LIN {X 0,Y 362,Z 148.389,A -85,B 0,C 180,E1 -12973.899,E2 -12973.899} C_VEL
LIN {X 0,Y 361.929,Z 148.396,A -85,B 0,C 180,E1 -12976.934,E2 -12976.934} C_VEL
LIN {X 0,Y 361.889,Z 148.404,A -85,B 0,C 180,E1 -12980.461,E2 -12980.461} C_VEL
LIN {X 0,Y 361.895,Z 148.403,A -85,B 0,C 180,E1 -12984.113,E2 -12984.113} C_VEL
LIN {X 0,Y 361.844,Z 148.41,A -85,B 0,C 180,E1 -12987.785,E2 -12987.785} C_VEL
LIN {X 0,Y 361.849,Z 148.409,A -85,B 0,C 180,E1 -12991.285,E2 -12991.285} C_VEL
LIN {X 0,Y 361.856,Z 148.405,A -85,B 0,C 180,E1 -12994.28,E2 -12994.28} C_VEL
LIN {X 0,Y 361.862,Z 148.405,A -85,B 0,C 180,E1 -12997.222,E2 -12997.222} C_VEL
LIN {X 0,Y 361.815,Z 148.415,A -85,B 0,C 180,E1 -13000.751,E2 -13000.751} C_VEL
LIN {X 0,Y 361.819,Z 148.419,A -85,B 0,C 180,E1 -13004.369,E2 -13004.369} C_VEL
LIN {X 0,Y 361.838,Z 148.415,A -85,B 0,C 180,E1 -13007.568,E2 -13007.568} C_VEL
LIN {X 0,Y 361.868,Z 148.41,A -85,B 0,C 180,E1 -13010.974,E2 -13010.974} C_VEL
LIN {X 0,Y 361.877,Z 148.405,A -85,B 0,C 180,E1 -13014.655,E2 -13014.655} C_VEL
LIN {X 0,Y 361.897,Z 148.548,A -85,B 0,C 180,E1 -13018.09,E2 -13018.09} C_VEL
LIN {X 0,Y 364.754,Z 160.107,A -85,B 0,C 180,E1 -13021.204,E2 -13021.204} C_VEL
LIN {X 0,Y 366.747,Z 170.569,A -85,B 0,C 180,E1 -13023.848,E2 -13023.848} C_VEL
LIN {X 0,Y 366.502,Z 174.041,A -85,B 0,C 180,E1 -13024.632,E2 -13024.632} C_VEL
LIN {X 0,Y 365.411,Z 184.836,A -85,B 0,C 180,E1 -13026.971,E2 -13026.971} C_VEL
LIN {X 0,Y 369.803,Z 207.145,A -85,B 0,C 180,E1 -13027.794,E2 -13027.794} C_VEL
LIN {X 0,Y 371.958,Z 222.29,A -85,B 0,C 180,E1 -13028.279,E2 -13028.279} C_VEL
LIN {X 0,Y 370.513,Z 294.23,A -85,B 0,C 180,E1 -13029.746,E2 -13029.746} C_VEL
LIN {X 0,Y 369.669,Z 307.871,A -85,B 0,C 180,E1 -13030.242,E2 -13030.242} C_VEL
LIN {X 0,Y 368.714,Z 319.646,A -85,B 0,C 180,E1 -13030.876,E2 -13030.876} C_VEL
LIN {X 0,Y 367.504,Z 331.641,A -85,B 0,C 180,E1 -13031.751,E2 -13031.751} C_VEL
LIN {X 0,Y 366.177,Z 343.107,A -85,B 0,C 180,E1 -13032.837,E2 -13032.837} C_VEL
LIN {X 0,Y 364.898,Z 353.468,A -85,B 0,C 180,E1 -13034.07,E2 -13034.07} C_VEL
LIN {X 0,Y 363.679,Z 362.827,A -85,B 0,C 180,E1 -13035.45,E2 -13035.45} C_VEL
LIN {X 0,Y 362.617,Z 371.909,A -85,B 0,C 180,E1 -13037.121,E2 -13037.121} C_VEL
LIN {X 0,Y 361.598,Z 379.26,A -85,B 0,C 180,E1 -13038.792,E2 -13038.792} C_VEL
LIN {X 0,Y 361.014,Z 385.178,A -85,B 0,C 180,E1 -13040.475,E2 -13040.475} C_VEL
LIN {X 0,Y 360.643,Z 389.866,A -85,B 0,C 180,E1 -13042.16,E2 -13042.16} C_VEL
LIN {X 0,Y 360.424,Z 393.696,A -85,B 0,C 180,E1 -13043.97,E2 -13043.97} C_VEL
LIN {X 0,Y 360.363,Z 396.045,A -85,B 0,C 180,E1 -13045.526,E2 -13045.526} C_VEL
LIN {X 0,Y 360.325,Z 397.269,A -85,B 0,C 180,E1 -13046.645,E2 -13046.645} C_VEL
LIN {X 0,Y 360.456,Z 398.443,A -85,B 0,C 180,E1 -13048.883,E2 -13048.883} C_VEL
LIN {X 0,Y 360.482,Z 398.443,A -85,B 0,C 180,E1 -13050,E2 -13050} C_VEL
LIN {X 0,Y 360.477,Z 398.05,A -85,B 0,C 180,E1 -13051.117,E2 -13051.117} C_VEL
LIN {X 0,Y 360.392,Z 397.212,A -85,B 0,C 180,E1 -13052.235,E2 -13052.235} C_VEL
LIN {X 0,Y 360.394,Z 394.304,A -85,B 0,C 180,E1 -13054.474,E2 -13054.474} C_VEL
LIN {X 0,Y 360.378,Z 391.384,A -85,B 0,C 180,E1 -13055.961,E2 -13055.961} C_VEL
LIN {X 0,Y 360.595,Z 386.495,A -85,B 0,C 180,E1 -13057.841,E2 -13057.841} C_VEL
LIN {X 0,Y 360.911,Z 380.822,A -85,B 0,C 180,E1 -13059.527,E2 -13059.527} C_VEL
LIN {X 0,Y 361.428,Z 373.709,A -85,B 0,C 180,E1 -13061.212,E2 -13061.212} C_VEL
LIN {X 0,Y 362.252,Z 364.807,A -85,B 0,C 180,E1 -13062.892,E2 -13062.892} C_VEL
LIN {X 0,Y 363.035,Z 356.181,A -85,B 0,C 180,E1 -13064.216,E2 -13064.216} C_VEL
LIN {X 0,Y 363.926,Z 345.713,A -85,B 0,C 180,E1 -13065.528,E2 -13065.528} C_VEL
LIN {X 0,Y 364.892,Z 334.368,A -85,B 0,C 180,E1 -13066.648,E2 -13066.648} C_VEL
LIN {X 0,Y 365.857,Z 321.79,A -85,B 0,C 180,E1 -13067.611,E2 -13067.611} C_VEL
LIN {X 0,Y 366.732,Z 308.962,A -85,B 0,C 180,E1 -13068.325,E2 -13068.325} C_VEL
LIN {X 0,Y 367.348,Z 295.296,A -85,B 0,C 180,E1 -13068.835,E2 -13068.835} C_VEL
LIN {X 0,Y 368.207,Z 245.144,A -85,B 0,C 180,E1 -13069.854,E2 -13069.854} C_VEL
LIN {X 0,Y 368.459,Z 220.259,A -85,B 0,C 180,E1 -13070.35,E2 -13070.35} C_VEL
LIN {X 0,Y 363.754,Z 185.456,A -85,B 0,C 180,E1 -13071.313,E2 -13071.313} C_VEL
LIN {X 0,Y 365.115,Z 169.471,A -85,B 0,C 180,E1 -13074.75,E2 -13074.75} C_VEL
LIN {X 0,Y 365.237,Z 165.158,A -85,B 0,C 180,E1 -13075.698,E2 -13075.698} C_VEL
LIN {X 0,Y 362.523,Z 151.236,A -85,B 0,C 180,E1 -13078.99,E2 -13078.99} C_VEL
LIN {X 0,Y 361.908,Z 148.408,A -85,B 0,C 180,E1 -13079.696,E2 -13079.696} C_VEL
LIN {X 0,Y 361.862,Z 148.407,A -85,B 0,C 180,E1 -13083.369,E2 -13083.369} C_VEL
LIN {X 0,Y 361.869,Z 148.406,A -85,B 0,C 180,E1 -13087.018,E2 -13087.018} C_VEL
LIN {X 0,Y 361.856,Z 148.413,A -85,B 0,C 180,E1 -13089.861,E2 -13089.861} C_VEL
LIN {X 0,Y 361.837,Z 148.41,A -85,B 0,C 180,E1 -13092.828,E2 -13092.828} C_VEL
LIN {X 0,Y 361.819,Z 148.415,A -85,B 0,C 180,E1 -13095.946,E2 -13095.946} C_VEL
LIN {X 0,Y 361.836,Z 148.412,A -85,B 0,C 180,E1 -13099.244,E2 -13099.244} C_VEL
LIN {X 0,Y 361.863,Z 148.407,A -85,B 0,C 180,E1 -13102.777,E2 -13102.777} C_VEL
LIN {X 0,Y 361.854,Z 148.411,A -85,B 0,C 180,E1 -13105.719,E2 -13105.719} C_VEL
LIN {X 0,Y 361.875,Z 148.408,A -85,B 0,C 180,E1 -13109.672,E2 -13109.672} C_VEL
LIN {X 0,Y 361.955,Z 148.399,A -85,B 0,C 180,E1 -13113.475,E2 -13113.475} C_VEL
LIN {X 0,Y 361.883,Z 148.41,A -85,B 0,C 180,E1 -13117.144,E2 -13117.144} C_VEL
LIN {X 0,Y 361.886,Z 148.406,A -85,B 0,C 180,E1 -13120.722,E2 -13120.722} C_VEL
LIN {X 0,Y 361.943,Z 148.396,A -85,B 0,C 180,E1 -13124.226,E2 -13124.226} C_VEL
LIN {X 0,Y 361.999,Z 148.391,A -85,B 0,C 180,E1 -13126.528,E2 -13126.528} C_VEL
LIN {X 0,Y 362,Z 148.389,A -85,B 0,C 180,E1 -13129.937,E2 -13129.937} C_VEL
LIN {X 0,Y 362.135,Z 148.374,A -85,B 0,C 180,E1 -13133.313,E2 -13133.313} C_VEL
LIN {X 0,Y 362.281,Z 148.354,A -85,B 0,C 180,E1 -13137.776,E2 -13137.776} C_VEL
LIN {X 0,Y 362.426,Z 148.337,A -85,B 0,C 180,E1 -13140,E2 -13140} C_VEL
LIN {X 0,Y 362.282,Z 148.356,A -85,B 0,C 180,E1 -13142.223,E2 -13142.223} C_VEL
LIN {X 0,Y 362.16,Z 148.374,A -85,B 0,C 180,E1 -13146.686,E2 -13146.686} C_VEL
LIN {X 0,Y 362.031,Z 148.388,A -85,B 0,C 180,E1 -13150.062,E2 -13150.062} C_VEL
LIN {X 0,Y 361.997,Z 148.391,A -85,B 0,C 180,E1 -13153.899,E2 -13153.899} C_VEL
LIN {X 0,Y 361.966,Z 148.396,A -85,B 0,C 180,E1 -13157.938,E2 -13157.938} C_VEL
LIN {X 0,Y 361.861,Z 148.408,A -85,B 0,C 180,E1 -13161.655,E2 -13161.655} C_VEL
LIN {X 0,Y 361.926,Z 148.399,A -85,B 0,C 180,E1 -13165.29,E2 -13165.29} C_VEL
LIN {X 0,Y 361.907,Z 148.404,A -85,B 0,C 180,E1 -13167.779,E2 -13167.779} C_VEL
LIN {X 0,Y 361.837,Z 148.412,A -85,B 0,C 180,E1 -13171.629,E2 -13171.629} C_VEL
LIN {X 0,Y 361.873,Z 148.406,A -85,B 0,C 180,E1 -13175.345,E2 -13175.345} C_VEL
LIN {X 0,Y 361.869,Z 148.406,A -85,B 0,C 180,E1 -13179.027,E2 -13179.027} C_VEL
LIN {X 0,Y 361.835,Z 148.41,A -85,B 0,C 180,E1 -13182.829,E2 -13182.829} C_VEL
LIN {X 0,Y 361.817,Z 148.415,A -85,B 0,C 180,E1 -13185.947,E2 -13185.947} C_VEL
LIN {X 0,Y 361.834,Z 148.413,A -85,B 0,C 180,E1 -13189.245,E2 -13189.245} C_VEL
LIN {X 0,Y 361.862,Z 148.407,A -85,B 0,C 180,E1 -13192.777,E2 -13192.777} C_VEL
LIN {X 0,Y 361.853,Z 148.411,A -85,B 0,C 180,E1 -13195.72,E2 -13195.72} C_VEL
LIN {X 0,Y 361.874,Z 148.408,A -85,B 0,C 180,E1 -13199.672,E2 -13199.672} C_VEL
LIN {X 0,Y 361.954,Z 148.399,A -85,B 0,C 180,E1 -13203.475,E2 -13203.475} C_VEL
LIN {X 0,Y 361.882,Z 148.41,A -85,B 0,C 180,E1 -13207.144,E2 -13207.144} C_VEL
LIN {X 0,Y 361.885,Z 148.406,A -85,B 0,C 180,E1 -13210.722,E2 -13210.722} C_VEL
LIN {X 0,Y 361.943,Z 148.397,A -85,B 0,C 180,E1 -13214.226,E2 -13214.226} C_VEL
LIN {X 0,Y 361.999,Z 148.392,A -85,B 0,C 180,E1 -13216.528,E2 -13216.528} C_VEL
LIN {X 0,Y 362,Z 148.389,A -85,B 0,C 180,E1 -13219.937,E2 -13219.937} C_VEL
LIN {X 0,Y 362.135,Z 148.374,A -85,B 0,C 180,E1 -13223.313,E2 -13223.313} C_VEL
LIN {X 0,Y 362.171,Z 148.447,A -85,B 0,C 180,E1 -13227.08,E2 -13227.08} C_VEL
LIN {X 0,Y 363.379,Z 154.733,A -85,B 0,C 180,E1 -13228.771,E2 -13228.771} C_VEL
LIN {X 0,Y 366.752,Z 166.026,A -85,B 0,C 180,E1 -13229.179,E2 -13229.179} C_VEL
LIN {X 0,Y 369.104,Z 178.936,A -85,B 0,C 180,E1 -13229.56,E2 -13229.56} C_VEL
LIN {X 0,Y 367.632,Z 262.636,A -85,B 0,C 180,E1 -13231.233,E2 -13231.233} C_VEL
LIN {X 0,Y 367.191,Z 276.354,A -85,B 0,C 180,E1 -13231.748,E2 -13231.748} C_VEL
LIN {X 0,Y 366.675,Z 288.171,A -85,B 0,C 180,E1 -13232.403,E2 -13232.403} C_VEL
LIN {X 0,Y 365.891,Z 300.242,A -85,B 0,C 180,E1 -13233.304,E2 -13233.304} C_VEL
LIN {X 0,Y 365.039,Z 311.767,A -85,B 0,C 180,E1 -13234.417,E2 -13234.417} C_VEL
LIN {X 0,Y 364.12,Z 322.178,A -85,B 0,C 180,E1 -13235.677,E2 -13235.677} C_VEL
LIN {X 0,Y 363.128,Z 332.343,A -85,B 0,C 180,E1 -13237.227,E2 -13237.227} C_VEL
LIN {X 0,Y 362.301,Z 341.262,A -85,B 0,C 180,E1 -13238.928,E2 -13238.928} C_VEL
LIN {X 0,Y 361.648,Z 348.361,A -85,B 0,C 180,E1 -13240.639,E2 -13240.639} C_VEL
LIN {X 0,Y 361.152,Z 354.036,A -85,B 0,C 180,E1 -13242.361,E2 -13242.361} C_VEL
LIN {X 0,Y 360.805,Z 358.477,A -85,B 0,C 180,E1 -13244.092,E2 -13244.092} C_VEL
LIN {X 0,Y 360.509,Z 361.81,A -85,B 0,C 180,E1 -13245.839,E2 -13245.839} C_VEL
LIN {X 0,Y 360.358,Z 363.616,A -85,B 0,C 180,E1 -13247.131,E2 -13247.131} C_VEL
LIN {X 0,Y 360.286,Z 364.645,A -85,B 0,C 180,E1 -13248.186,E2 -13248.186} C_VEL
LIN {X 0,Y 360.274,Z 365.465,A -85,B 0,C 180,E1 -13249.708,E2 -13249.708} C_VEL
LIN {X 0,Y 360.311,Z 365.692,A -85,B 0,C 180,E1 -13250.568,E2 -13250.568} C_VEL
LIN {X 0,Y 360.34,Z 365.549,A -85,B 0,C 180,E1 -13251.751,E2 -13251.751} C_VEL
LIN {X 0,Y 360.522,Z 364.413,A -85,B 0,C 180,E1 -13253.621,E2 -13253.621} C_VEL
LIN {X 0,Y 360.663,Z 363.388,A -85,B 0,C 180,E1 -13254.55,E2 -13254.55} C_VEL
LIN {X 0,Y 360.166,Z 362.258,A -85,B 0,C 180,E1 -13255.467,E2 -13255.467} C_VEL
LIN {X 0,Y 357.686,Z 359.944,A -85,B 0,C 180,E1 -13256.956,E2 -13256.956} C_VEL
LIN {X 0,Y 355.646,Z 357.657,A -85,B 0,C 180,E1 -13258.138,E2 -13258.138} C_VEL
LIN {X 0,Y 354.922,Z 355.563,A -85,B 0,C 180,E1 -13259.026,E2 -13259.026} C_VEL
LIN {X 0,Y 354.946,Z 354.762,A -85,B 0,C 180,E1 -13259.319,E2 -13259.319} C_VEL
LIN {X 0,Y 355.694,Z 349.778,A -85,B 0,C 180,E1 -13260.912,E2 -13260.912} C_VEL
LIN {X 0,Y 356.802,Z 342.363,A -85,B 0,C 180,E1 -13262.798,E2 -13262.798} C_VEL
LIN {X 0,Y 358.029,Z 334.009,A -85,B 0,C 180,E1 -13264.468,E2 -13264.468} C_VEL
LIN {X 0,Y 359.219,Z 324.905,A -85,B 0,C 180,E1 -13265.94,E2 -13265.94} C_VEL
LIN {X 0,Y 360.637,Z 314.081,A -85,B 0,C 180,E1 -13267.341,E2 -13267.341} C_VEL
LIN {X 0,Y 362.038,Z 302.196,A -85,B 0,C 180,E1 -13268.534,E2 -13268.534} C_VEL
LIN {X 0,Y 363.121,Z 289.635,A -85,B 0,C 180,E1 -13269.515,E2 -13269.515} C_VEL
LIN {X 0,Y 363.912,Z 277.193,A -85,B 0,C 180,E1 -13270.223,E2 -13270.223} C_VEL
LIN {X 0,Y 364.539,Z 263.315,A -85,B 0,C 180,E1 -13270.752,E2 -13270.752} C_VEL
LIN {X 0,Y 366.444,Z 181.628,A -85,B 0,C 180,E1 -13272.428,E2 -13272.428} C_VEL
LIN {X 0,Y 365.137,Z 176.337,A -85,B 0,C 180,E1 -13272.647,E2 -13272.647} C_VEL
LIN {X 0,Y 357.636,Z 158.854,A -85,B 0,C 180,E1 -13273.66,E2 -13273.66} C_VEL
LIN {X 0,Y 356.429,Z 155.986,A -85,B 0,C 180,E1 -13273.846,E2 -13273.846} C_VEL
LIN {X 0,Y 354.78,Z 149.298,A -85,B 0,C 180,E1 -13275.91,E2 -13275.91} C_VEL
LIN {X 0,Y 354.765,Z 149.297,A -85,B 0,C 180,E1 -13279.176,E2 -13279.176} C_VEL
LIN {X 0,Y 354.799,Z 149.289,A -85,B 0,C 180,E1 -13282.405,E2 -13282.405} C_VEL
LIN {X 0,Y 354.808,Z 149.288,A -85,B 0,C 180,E1 -13284.941,E2 -13284.941} C_VEL
LIN {X 0,Y 354.793,Z 149.292,A -85,B 0,C 180,E1 -13288.406,E2 -13288.406} C_VEL
LIN {X 0,Y 354.797,Z 149.289,A -85,B 0,C 180,E1 -13291.615,E2 -13291.615} C_VEL
LIN {X 0,Y 354.804,Z 149.29,A -85,B 0,C 180,E1 -13295.42,E2 -13295.42} C_VEL
LIN {X 0,Y 354.816,Z 149.288,A -85,B 0,C 180,E1 -13299.113,E2 -13299.113} C_VEL
LIN {X 0,Y 354.837,Z 149.287,A -85,B 0,C 180,E1 -13302.717,E2 -13302.717} C_VEL
LIN {X 0,Y 354.909,Z 149.274,A -85,B 0,C 180,E1 -13306.254,E2 -13306.254} C_VEL
LIN {X 0,Y 354.949,Z 149.262,A -85,B 0,C 180,E1 -13309.735,E2 -13309.735} C_VEL
LIN {X 0,Y 355.088,Z 149.245,A -85,B 0,C 180,E1 -13313.18,E2 -13313.18} C_VEL
LIN {X 0,Y 355.22,Z 149.228,A -85,B 0,C 180,E1 -13317.732,E2 -13317.732} C_VEL
LIN {X 0,Y 355.146,Z 149.244,A -85,B 0,C 180,E1 -13321.134,E2 -13321.134} C_VEL
LIN {X 0,Y 355.227,Z 149.225,A -85,B 0,C 180,E1 -13322.268,E2 -13322.268} C_VEL
LIN {X 0,Y 355.089,Z 149.248,A -85,B 0,C 180,E1 -13326.82,E2 -13326.82} C_VEL
LIN {X 0,Y 354.956,Z 149.269,A -85,B 0,C 180,E1 -13330.265,E2 -13330.265} C_VEL
LIN {X 0,Y 354.945,Z 149.269,A -85,B 0,C 180,E1 -13334.019,E2 -13334.019} C_VEL
LIN {X 0,Y 354.892,Z 149.269,A -85,B 0,C 180,E1 -13338.092,E2 -13338.092} C_VEL
LIN {X 0,Y 354.821,Z 149.279,A -85,B 0,C 180,E1 -13341.418,E2 -13341.418} C_VEL
LIN {X 0,Y 354.851,Z 149.282,A -85,B 0,C 180,E1 -13344.577,E2 -13344.577} C_VEL
LIN {X 0,Y 354.802,Z 149.288,A -85,B 0,C 180,E1 -13348.386,E2 -13348.386} C_VEL
LIN {X 0,Y 354.789,Z 149.29,A -85,B 0,C 180,E1 -13352.333,E2 -13352.333} C_VEL
LIN {X 0,Y 354.824,Z 149.286,A -85,B 0,C 180,E1 -13355.699,E2 -13355.699} C_VEL
LIN {X 0,Y 354.77,Z 149.293,A -85,B 0,C 180,E1 -13359.413,E2 -13359.413} C_VEL
LIN {X 0,Y 354.787,Z 149.291,A -85,B 0,C 180,E1 -13362.867,E2 -13362.867} C_VEL
LIN {X 0,Y 354.769,Z 149.294,A -85,B 0,C 180,E1 -13366.104,E2 -13366.104} C_VEL
LIN {X 0,Y 354.788,Z 149.293,A -85,B 0,C 180,E1 -13369.179,E2 -13369.179} C_VEL
LIN {X 0,Y 354.808,Z 149.281,A -85,B 0,C 180,E1 -13372.403,E2 -13372.403} C_VEL
LIN {X 0,Y 354.814,Z 149.283,A -85,B 0,C 180,E1 -13374.941,E2 -13374.941} C_VEL
LIN {X 0,Y 354.841,Z 149.47,A -85,B 0,C 180,E1 -13377.588,E2 -13377.588} C_VEL
LIN {X 0,Y 357.879,Z 161.515,A -85,B 0,C 180,E1 -13380.92,E2 -13380.92} C_VEL
LIN {X 0,Y 359.925,Z 172.344,A -85,B 0,C 180,E1 -13383.718,E2 -13383.718} C_VEL
LIN {X 0,Y 358.686,Z 184.194,A -85,B 0,C 180,E1 -13386.412,E2 -13386.412} C_VEL
LIN {X 0,Y 363.396,Z 208.056,A -85,B 0,C 180,E1 -13387.327,E2 -13387.327} C_VEL
LIN {X 0,Y 365.533,Z 223.693,A -85,B 0,C 180,E1 -13387.835,E2 -13387.835} C_VEL
LIN {X 0,Y 364.043,Z 294.036,A -85,B 0,C 180,E1 -13389.296,E2 -13389.296} C_VEL
LIN {X 0,Y 363.162,Z 307.631,A -85,B 0,C 180,E1 -13389.799,E2 -13389.799} C_VEL
LIN {X 0,Y 362.112,Z 319.389,A -85,B 0,C 180,E1 -13390.44,E2 -13390.44} C_VEL
LIN {X 0,Y 360.948,Z 330.571,A -85,B 0,C 180,E1 -13391.26,E2 -13391.26} C_VEL
LIN {X 0,Y 359.569,Z 342.172,A -85,B 0,C 180,E1 -13392.364,E2 -13392.364} C_VEL
LIN {X 0,Y 358.176,Z 352.638,A -85,B 0,C 180,E1 -13393.617,E2 -13393.617} C_VEL
LIN {X 0,Y 357.081,Z 360.972,A -85,B 0,C 180,E1 -13394.843,E2 -13394.843} C_VEL
LIN {X 0,Y 356.081,Z 369.153,A -85,B 0,C 180,E1 -13396.299,E2 -13396.299} C_VEL
LIN {X 0,Y 354.91,Z 376.956,A -85,B 0,C 180,E1 -13397.999,E2 -13397.999} C_VEL
LIN {X 0,Y 354.186,Z 383.231,A -85,B 0,C 180,E1 -13399.712,E2 -13399.712} C_VEL
LIN {X 0,Y 353.691,Z 388.249,A -85,B 0,C 180,E1 -13401.429,E2 -13401.429} C_VEL
LIN {X 0,Y 353.397,Z 392.158,A -85,B 0,C 180,E1 -13403.147,E2 -13403.147} C_VEL
LIN {X 0,Y 353.274,Z 395.798,A -85,B 0,C 180,E1 -13405.436,E2 -13405.436} C_VEL
LIN {X 0,Y 353.244,Z 396.993,A -85,B 0,C 180,E1 -13406.578,E2 -13406.578} C_VEL
LIN {X 0,Y 353.358,Z 398.126,A -85,B 0,C 180,E1 -13408.86,E2 -13408.86} C_VEL
LIN {X 0,Y 353.4,Z 398.109,A -85,B 0,C 180,E1 -13410,E2 -13410} C_VEL
LIN {X 0,Y 353.38,Z 397.69,A -85,B 0,C 180,E1 -13411.139,E2 -13411.139} C_VEL
LIN {X 0,Y 353.294,Z 396.823,A -85,B 0,C 180,E1 -13412.28,E2 -13412.28} C_VEL
LIN {X 0,Y 353.261,Z 395.554,A -85,B 0,C 180,E1 -13413.421,E2 -13413.421} C_VEL
LIN {X 0,Y 353.261,Z 392.846,A -85,B 0,C 180,E1 -13415.136,E2 -13415.136} C_VEL
LIN {X 0,Y 353.353,Z 389.096,A -85,B 0,C 180,E1 -13416.854,E2 -13416.854} C_VEL
LIN {X 0,Y 353.625,Z 384.206,A -85,B 0,C 180,E1 -13418.572,E2 -13418.572} C_VEL
LIN {X 0,Y 354.033,Z 378.023,A -85,B 0,C 180,E1 -13420.292,E2 -13420.292} C_VEL
LIN {X 0,Y 354.733,Z 370.329,A -85,B 0,C 180,E1 -13422.007,E2 -13422.007} C_VEL
LIN {X 0,Y 355.417,Z 362.431,A -85,B 0,C 180,E1 -13423.435,E2 -13423.435} C_VEL
LIN {X 0,Y 356.248,Z 352.768,A -85,B 0,C 180,E1 -13424.86,E2 -13424.86} C_VEL
LIN {X 0,Y 357.25,Z 342.056,A -85,B 0,C 180,E1 -13426.133,E2 -13426.133} C_VEL
LIN {X 0,Y 358.193,Z 331.718,A -85,B 0,C 180,E1 -13427.116,E2 -13427.116} C_VEL
LIN {X 0,Y 359.114,Z 319.397,A -85,B 0,C 180,E1 -13428.026,E2 -13428.026} C_VEL
LIN {X 0,Y 360.056,Z 305.712,A -85,B 0,C 180,E1 -13428.751,E2 -13428.751} C_VEL
LIN {X 0,Y 360.599,Z 292.723,A -85,B 0,C 180,E1 -13429.201,E2 -13429.201} C_VEL
LIN {X 0,Y 361.667,Z 221.058,A -85,B 0,C 180,E1 -13430.656,E2 -13430.656} C_VEL
LIN {X 0,Y 356.802,Z 185.169,A -85,B 0,C 180,E1 -13431.664,E2 -13431.664} C_VEL
LIN {X 0,Y 358.188,Z 170.181,A -85,B 0,C 180,E1 -13434.951,E2 -13434.951} C_VEL
LIN {X 0,Y 358.22,Z 166.044,A -85,B 0,C 180,E1 -13435.882,E2 -13435.882} C_VEL
LIN {X 0,Y 355.722,Z 153.285,A -85,B 0,C 180,E1 -13438.95,E2 -13438.95} C_VEL
LIN {X 0,Y 354.85,Z 149.286,A -85,B 0,C 180,E1 -13439.965,E2 -13439.965} C_VEL
LIN {X 0,Y 354.807,Z 149.289,A -85,B 0,C 180,E1 -13443.702,E2 -13443.702} C_VEL
LIN {X 0,Y 354.799,Z 149.288,A -85,B 0,C 180,E1 -13446.459,E2 -13446.459} C_VEL
LIN {X 0,Y 354.825,Z 149.285,A -85,B 0,C 180,E1 -13449.423,E2 -13449.423} C_VEL
LIN {X 0,Y 354.789,Z 149.288,A -85,B 0,C 180,E1 -13452.867,E2 -13452.867} C_VEL
LIN {X 0,Y 354.768,Z 149.292,A -85,B 0,C 180,E1 -13456.103,E2 -13456.103} C_VEL
LIN {X 0,Y 354.788,Z 149.29,A -85,B 0,C 180,E1 -13459.179,E2 -13459.179} C_VEL
LIN {X 0,Y 354.807,Z 149.285,A -85,B 0,C 180,E1 -13462.402,E2 -13462.402} C_VEL
LIN {X 0,Y 354.812,Z 149.286,A -85,B 0,C 180,E1 -13464.94,E2 -13464.94} C_VEL
LIN {X 0,Y 354.793,Z 149.287,A -85,B 0,C 180,E1 -13468.405,E2 -13468.405} C_VEL
LIN {X 0,Y 354.851,Z 149.283,A -85,B 0,C 180,E1 -13471.619,E2 -13471.619} C_VEL
LIN {X 0,Y 354.899,Z 149.274,A -85,B 0,C 180,E1 -13474.172,E2 -13474.172} C_VEL
LIN {X 0,Y 354.817,Z 149.285,A -85,B 0,C 180,E1 -13477.893,E2 -13477.893} C_VEL
LIN {X 0,Y 354.889,Z 149.275,A -85,B 0,C 180,E1 -13481.908,E2 -13481.908} C_VEL
LIN {X 0,Y 354.943,Z 149.268,A -85,B 0,C 180,E1 -13485.981,E2 -13485.981} C_VEL
LIN {X 0,Y 354.956,Z 149.267,A -85,B 0,C 180,E1 -13489.735,E2 -13489.735} C_VEL
LIN {X 0,Y 355.098,Z 149.252,A -85,B 0,C 180,E1 -13493.18,E2 -13493.18} C_VEL
LIN {X 0,Y 355.244,Z 149.231,A -85,B 0,C 180,E1 -13497.732,E2 -13497.732} C_VEL
LIN {X 0,Y 355.396,Z 149.213,A -85,B 0,C 180,E1 -13500,E2 -13500} C_VEL
LIN {X 0,Y 355.245,Z 149.233,A -85,B 0,C 180,E1 -13502.267,E2 -13502.267} C_VEL
LIN {X 0,Y 355.124,Z 149.249,A -85,B 0,C 180,E1 -13506.819,E2 -13506.819} C_VEL
LIN {X 0,Y 354.977,Z 149.268,A -85,B 0,C 180,E1 -13510.264,E2 -13510.264} C_VEL
LIN {X 0,Y 354.942,Z 149.271,A -85,B 0,C 180,E1 -13514.019,E2 -13514.019} C_VEL
LIN {X 0,Y 354.922,Z 149.275,A -85,B 0,C 180,E1 -13518.108,E2 -13518.108} C_VEL
LIN {X 0,Y 354.816,Z 149.29,A -85,B 0,C 180,E1 -13522.107,E2 -13522.107} C_VEL
LIN {X 0,Y 354.897,Z 149.277,A -85,B 0,C 180,E1 -13525.827,E2 -13525.827} C_VEL
LIN {X 0,Y 354.816,Z 149.287,A -85,B 0,C 180,E1 -13529.682,E2 -13529.682} C_VEL
LIN {X 0,Y 354.805,Z 149.289,A -85,B 0,C 180,E1 -13533.702,E2 -13533.702} C_VEL
LIN {X 0,Y 354.797,Z 149.288,A -85,B 0,C 180,E1 -13536.459,E2 -13536.459} C_VEL
LIN {X 0,Y 354.823,Z 149.286,A -85,B 0,C 180,E1 -13539.424,E2 -13539.424} C_VEL
LIN {X 0,Y 354.787,Z 149.288,A -85,B 0,C 180,E1 -13542.867,E2 -13542.867} C_VEL
LIN {X 0,Y 354.766,Z 149.292,A -85,B 0,C 180,E1 -13546.104,E2 -13546.104} C_VEL
LIN {X 0,Y 354.786,Z 149.29,A -85,B 0,C 180,E1 -13549.179,E2 -13549.179} C_VEL
LIN {X 0,Y 354.805,Z 149.286,A -85,B 0,C 180,E1 -13552.403,E2 -13552.403} C_VEL
LIN {X 0,Y 354.811,Z 149.286,A -85,B 0,C 180,E1 -13554.941,E2 -13554.941} C_VEL
LIN {X 0,Y 354.792,Z 149.287,A -85,B 0,C 180,E1 -13558.405,E2 -13558.405} C_VEL
LIN {X 0,Y 354.85,Z 149.283,A -85,B 0,C 180,E1 -13561.619,E2 -13561.619} C_VEL
LIN {X 0,Y 354.898,Z 149.274,A -85,B 0,C 180,E1 -13564.173,E2 -13564.173} C_VEL
LIN {X 0,Y 354.816,Z 149.285,A -85,B 0,C 180,E1 -13567.893,E2 -13567.893} C_VEL
LIN {X 0,Y 354.889,Z 149.275,A -85,B 0,C 180,E1 -13571.908,E2 -13571.908} C_VEL
LIN {X 0,Y 354.942,Z 149.268,A -85,B 0,C 180,E1 -13575.981,E2 -13575.981} C_VEL
LIN {X 0,Y 354.956,Z 149.267,A -85,B 0,C 180,E1 -13579.735,E2 -13579.735} C_VEL
LIN {X 0,Y 355.099,Z 149.251,A -85,B 0,C 180,E1 -13583.18,E2 -13583.18} C_VEL
LIN {X 0,Y 355.066,Z 149.352,A -85,B 0,C 180,E1 -13586.844,E2 -13586.844} C_VEL
LIN {X 0,Y 356.261,Z 155.044,A -85,B 0,C 180,E1 -13588.403,E2 -13588.403} C_VEL
LIN {X 0,Y 360.144,Z 167.706,A -85,B 0,C 180,E1 -13588.882,E2 -13588.882} C_VEL
LIN {X 0,Y 362.358,Z 180.442,A -85,B 0,C 180,E1 -13589.261,E2 -13589.261} C_VEL
LIN {X 0,Y 360.819,Z 262.013,A -85,B 0,C 180,E1 -13590.907,E2 -13590.907} C_VEL
LIN {X 0,Y 360.357,Z 275.325,A -85,B 0,C 180,E1 -13591.397,E2 -13591.397} C_VEL
LIN {X 0,Y 359.831,Z 288.034,A -85,B 0,C 180,E1 -13592.099,E2 -13592.099} C_VEL
LIN {X 0,Y 359.101,Z 299.522,A -85,B 0,C 180,E1 -13592.953,E2 -13592.953} C_VEL
LIN {X 0,Y 358.203,Z 311.181,A -85,B 0,C 180,E1 -13594.079,E2 -13594.079} C_VEL
LIN {X 0,Y 357.226,Z 321.772,A -85,B 0,C 180,E1 -13595.362,E2 -13595.362} C_VEL
LIN {X 0,Y 356.316,Z 331.265,A -85,B 0,C 180,E1 -13596.797,E2 -13596.797} C_VEL
LIN {X 0,Y 355.484,Z 339.743,A -85,B 0,C 180,E1 -13598.385,E2 -13598.385} C_VEL
LIN {X 0,Y 354.772,Z 346.67,A -85,B 0,C 180,E1 -13599.982,E2 -13599.982} C_VEL
LIN {X 0,Y 354.297,Z 351.844,A -85,B 0,C 180,E1 -13601.442,E2 -13601.442} C_VEL
LIN {X 0,Y 353.874,Z 357.114,A -85,B 0,C 180,E1 -13603.308,E2 -13603.308} C_VEL
LIN {X 0,Y 353.544,Z 360.697,A -85,B 0,C 180,E1 -13604.977,E2 -13604.977} C_VEL
LIN {X 0,Y 353.383,Z 362.683,A -85,B 0,C 180,E1 -13606.167,E2 -13606.167} C_VEL
LIN {X 0,Y 353.266,Z 364.17,A -85,B 0,C 180,E1 -13607.363,E2 -13607.363} C_VEL
LIN {X 0,Y 353.197,Z 365.221,A -85,B 0,C 180,E1 -13608.565,E2 -13608.565} C_VEL
LIN {X 0,Y 353.219,Z 366.034,A -85,B 0,C 180,E1 -13610.746,E2 -13610.746} C_VEL
LIN {X 0,Y 353.304,Z 365.733,A -85,B 0,C 180,E1 -13612.207,E2 -13612.207} C_VEL
LIN {X 0,Y 353.468,Z 364.656,A -85,B 0,C 180,E1 -13613.849,E2 -13613.849} C_VEL
LIN {X 0,Y 353.878,Z 362.116,A -85,B 0,C 180,E1 -13615.908,E2 -13615.908} C_VEL
LIN {X 0,Y 354.394,Z 358.612,A -85,B 0,C 180,E1 -13617.777,E2 -13617.777} C_VEL
LIN {X 0,Y 354.946,Z 354.762,A -85,B 0,C 180,E1 -13619.319,E2 -13619.319} C_VEL
LIN {X 0,Y 354.642,Z 352.319,A -85,B 0,C 180,E1 -13620.186,E2 -13620.186} C_VEL
LIN {X 0,Y 352.518,Z 348.05,A -85,B 0,C 180,E1 -13621.596,E2 -13621.596} C_VEL
LIN {X 0,Y 350.513,Z 343.223,A -85,B 0,C 180,E1 -13622.966,E2 -13622.966} C_VEL
LIN {X 0,Y 350.392,Z 339.816,A -85,B 0,C 180,E1 -13623.76,E2 -13623.76} C_VEL
LIN {X 0,Y 351.762,Z 331.061,A -85,B 0,C 180,E1 -13625.409,E2 -13625.409} C_VEL
LIN {X 0,Y 353.1,Z 321.252,A -85,B 0,C 180,E1 -13626.891,E2 -13626.891} C_VEL
LIN {X 0,Y 354.431,Z 311.198,A -85,B 0,C 180,E1 -13628.11,E2 -13628.11} C_VEL
LIN {X 0,Y 355.766,Z 299.812,A -85,B 0,C 180,E1 -13629.209,E2 -13629.209} C_VEL
LIN {X 0,Y 356.755,Z 287.761,A -85,B 0,C 180,E1 -13630.107,E2 -13630.107} C_VEL
LIN {X 0,Y 357.635,Z 274.984,A -85,B 0,C 180,E1 -13630.799,E2 -13630.799} C_VEL
LIN {X 0,Y 358.167,Z 262.187,A -85,B 0,C 180,E1 -13631.261,E2 -13631.261} C_VEL
LIN {X 0,Y 359.955,Z 182.211,A -85,B 0,C 180,E1 -13632.931,E2 -13632.931} C_VEL
LIN {X 0,Y 358.739,Z 178.019,A -85,B 0,C 180,E1 -13633.128,E2 -13633.128} C_VEL
LIN {X 0,Y 351.768,Z 161.902,A -85,B 0,C 180,E1 -13634.105,E2 -13634.105} C_VEL
LIN {X 0,Y 349.223,Z 156.335,A -85,B 0,C 180,E1 -13634.489,E2 -13634.489} C_VEL
LIN {X 0,Y 347.72,Z 150.179,A -85,B 0,C 180,E1 -13636.442,E2 -13636.442} C_VEL
LIN {X 0,Y 347.697,Z 150.171,A -85,B 0,C 180,E1 -13639.698,E2 -13639.698} C_VEL
LIN {X 0,Y 347.755,Z 150.162,A -85,B 0,C 180,E1 -13642.679,E2 -13642.679} C_VEL
LIN {X 0,Y 347.748,Z 150.168,A -85,B 0,C 180,E1 -13645.957,E2 -13645.957} C_VEL
LIN {X 0,Y 347.738,Z 150.172,A -85,B 0,C 180,E1 -13649.651,E2 -13649.651} C_VEL
LIN {X 0,Y 347.734,Z 150.17,A -85,B 0,C 180,E1 -13653.6,E2 -13653.6} C_VEL
LIN {X 0,Y 347.746,Z 150.171,A -85,B 0,C 180,E1 -13656.159,E2 -13656.159} C_VEL
LIN {X 0,Y 347.763,Z 150.167,A -85,B 0,C 180,E1 -13659.907,E2 -13659.907} C_VEL
LIN {X 0,Y 347.782,Z 150.163,A -85,B 0,C 180,E1 -13663.566,E2 -13663.566} C_VEL
LIN {X 0,Y 347.864,Z 150.152,A -85,B 0,C 180,E1 -13667.16,E2 -13667.16} C_VEL
LIN {X 0,Y 347.934,Z 150.144,A -85,B 0,C 180,E1 -13670.701,E2 -13670.701} C_VEL
LIN {X 0,Y 348.037,Z 150.124,A -85,B 0,C 180,E1 -13674.205,E2 -13674.205} C_VEL
LIN {X 0,Y 348.181,Z 150.105,A -85,B 0,C 180,E1 -13677.687,E2 -13677.687} C_VEL
LIN {X 0,Y 348.117,Z 150.119,A -85,B 0,C 180,E1 -13681.157,E2 -13681.157} C_VEL
LIN {X 0,Y 348.188,Z 150.102,A -85,B 0,C 180,E1 -13682.314,E2 -13682.314} C_VEL
LIN {X 0,Y 348.056,Z 150.125,A -85,B 0,C 180,E1 -13686.959,E2 -13686.959} C_VEL
LIN {X 0,Y 347.897,Z 150.148,A -85,B 0,C 180,E1 -13690.476,E2 -13690.476} C_VEL
LIN {X 0,Y 347.901,Z 150.146,A -85,B 0,C 180,E1 -13694.15,E2 -13694.15} C_VEL
LIN {X 0,Y 347.831,Z 150.149,A -85,B 0,C 180,E1 -13698.259,E2 -13698.259} C_VEL
LIN {X 0,Y 347.771,Z 150.155,A -85,B 0,C 180,E1 -13701.627,E2 -13701.627} C_VEL
LIN {X 0,Y 347.771,Z 150.163,A -85,B 0,C 180,E1 -13705.112,E2 -13705.112} C_VEL
LIN {X 0,Y 347.748,Z 150.168,A -85,B 0,C 180,E1 -13709.015,E2 -13709.015} C_VEL
LIN {X 0,Y 347.741,Z 150.167,A -85,B 0,C 180,E1 -13711.914,E2 -13711.914} C_VEL
LIN {X 0,Y 347.79,Z 150.162,A -85,B 0,C 180,E1 -13715.875,E2 -13715.875} C_VEL
LIN {X 0,Y 347.733,Z 150.173,A -85,B 0,C 180,E1 -13718.796,E2 -13718.796} C_VEL
LIN {X 0,Y 347.746,Z 150.17,A -85,B 0,C 180,E1 -13721.831,E2 -13721.831} C_VEL
LIN {X 0,Y 347.708,Z 150.175,A -85,B 0,C 180,E1 -13725.027,E2 -13725.027} C_VEL
LIN {X 0,Y 347.752,Z 150.17,A -85,B 0,C 180,E1 -13728.397,E2 -13728.397} C_VEL
LIN {X 0,Y 347.774,Z 150.159,A -85,B 0,C 180,E1 -13732.012,E2 -13732.012} C_VEL
LIN {X 0,Y 347.747,Z 150.163,A -85,B 0,C 180,E1 -13735.536,E2 -13735.536} C_VEL
LIN {X 0,Y 347.779,Z 150.231,A -85,B 0,C 180,E1 -13737.003,E2 -13737.003} C_VEL
LIN {X 0,Y 350.944,Z 162.918,A -85,B 0,C 180,E1 -13740.617,E2 -13740.617} C_VEL
LIN {X 0,Y 352.954,Z 173.103,A -85,B 0,C 180,E1 -13743.321,E2 -13743.321} C_VEL
LIN {X 0,Y 352.964,Z 175.978,A -85,B 0,C 180,E1 -13744.02,E2 -13744.02} C_VEL
LIN {X 0,Y 352.012,Z 183.867,A -85,B 0,C 180,E1 -13745.841,E2 -13745.841} C_VEL
LIN {X 0,Y 356.953,Z 208.637,A -85,B 0,C 180,E1 -13746.832,E2 -13746.832} C_VEL
LIN {X 0,Y 359.157,Z 223.894,A -85,B 0,C 180,E1 -13747.35,E2 -13747.35} C_VEL
LIN {X 0,Y 357.595,Z 293.844,A -85,B 0,C 180,E1 -13748.83,E2 -13748.83} C_VEL
LIN {X 0,Y 356.673,Z 307.391,A -85,B 0,C 180,E1 -13749.339,E2 -13749.339} C_VEL
LIN {X 0,Y 355.473,Z 320.169,A -85,B 0,C 180,E1 -13750.059,E2 -13750.059} C_VEL
LIN {X 0,Y 354.113,Z 332.646,A -85,B 0,C 180,E1 -13751.035,E2 -13751.035} C_VEL
LIN {X 0,Y 352.665,Z 343.811,A -85,B 0,C 180,E1 -13752.158,E2 -13752.158} C_VEL
LIN {X 0,Y 351.248,Z 353.901,A -85,B 0,C 180,E1 -13753.434,E2 -13753.434} C_VEL
LIN {X 0,Y 349.941,Z 363.029,A -85,B 0,C 180,E1 -13754.865,E2 -13754.865} C_VEL
LIN {X 0,Y 348.743,Z 371.955,A -85,B 0,C 180,E1 -13756.6,E2 -13756.6} C_VEL
LIN {X 0,Y 347.624,Z 379.168,A -85,B 0,C 180,E1 -13758.336,E2 -13758.336} C_VEL
LIN {X 0,Y 346.969,Z 384.955,A -85,B 0,C 180,E1 -13760.086,E2 -13760.086} C_VEL
LIN {X 0,Y 346.517,Z 389.538,A -85,B 0,C 180,E1 -13761.838,E2 -13761.838} C_VEL
LIN {X 0,Y 346.235,Z 393.783,A -85,B 0,C 180,E1 -13764.056,E2 -13764.056} C_VEL
LIN {X 0,Y 346.17,Z 395.559,A -85,B 0,C 180,E1 -13765.342,E2 -13765.342} C_VEL
LIN {X 0,Y 346.165,Z 396.716,A -85,B 0,C 180,E1 -13766.508,E2 -13766.508} C_VEL
LIN {X 0,Y 346.259,Z 397.81,A -85,B 0,C 180,E1 -13768.837,E2 -13768.837} C_VEL
LIN {X 0,Y 346.321,Z 397.776,A -85,B 0,C 180,E1 -13770,E2 -13770} C_VEL
LIN {X 0,Y 346.284,Z 397.323,A -85,B 0,C 180,E1 -13771.163,E2 -13771.163} C_VEL
LIN {X 0,Y 346.182,Z 395.148,A -85,B 0,C 180,E1 -13773.492,E2 -13773.492} C_VEL
LIN {X 0,Y 346.173,Z 392.003,A -85,B 0,C 180,E1 -13775.457,E2 -13775.457} C_VEL
LIN {X 0,Y 346.371,Z 387.107,A -85,B 0,C 180,E1 -13777.578,E2 -13777.578} C_VEL
LIN {X 0,Y 346.751,Z 380.721,A -85,B 0,C 180,E1 -13779.626,E2 -13779.626} C_VEL
LIN {X 0,Y 347.289,Z 373.752,A -85,B 0,C 180,E1 -13781.379,E2 -13781.379} C_VEL
LIN {X 0,Y 348.046,Z 366.637,A -85,B 0,C 180,E1 -13782.833,E2 -13782.833} C_VEL
LIN {X 0,Y 348.93,Z 357.042,A -85,B 0,C 180,E1 -13784.431,E2 -13784.431} C_VEL
LIN {X 0,Y 349.814,Z 347.356,A -85,B 0,C 180,E1 -13785.737,E2 -13785.737} C_VEL
LIN {X 0,Y 350.832,Z 336.8,A -85,B 0,C 180,E1 -13786.886,E2 -13786.886} C_VEL
LIN {X 0,Y 351.804,Z 325.148,A -85,B 0,C 180,E1 -13787.887,E2 -13787.887} C_VEL
LIN {X 0,Y 352.724,Z 313.059,A -85,B 0,C 180,E1 -13788.665,E2 -13788.665} C_VEL
LIN {X 0,Y 353.509,Z 299.984,A -85,B 0,C 180,E1 -13789.262,E2 -13789.262} C_VEL
LIN {X 0,Y 353.878,Z 287.59,A -85,B 0,C 180,E1 -13789.618,E2 -13789.618} C_VEL
LIN {X 0,Y 354.826,Z 221.246,A -85,B 0,C 180,E1 -13790.978,E2 -13790.978} C_VEL
LIN {X 0,Y 349.886,Z 184.911,A -85,B 0,C 180,E1 -13792.023,E2 -13792.023} C_VEL
LIN {X 0,Y 351.317,Z 169.844,A -85,B 0,C 180,E1 -13795.386,E2 -13795.386} C_VEL
LIN {X 0,Y 350.851,Z 165.254,A -85,B 0,C 180,E1 -13796.468,E2 -13796.468} C_VEL
LIN {X 0,Y 348.538,Z 153.622,A -85,B 0,C 180,E1 -13799.34,E2 -13799.34} C_VEL
LIN {X 0,Y 347.808,Z 150.163,A -85,B 0,C 180,E1 -13800.253,E2 -13800.253} C_VEL
LIN {X 0,Y 347.746,Z 150.166,A -85,B 0,C 180,E1 -13804.464,E2 -13804.464} C_VEL
LIN {X 0,Y 347.775,Z 150.166,A -85,B 0,C 180,E1 -13807.988,E2 -13807.988} C_VEL
LIN {X 0,Y 347.752,Z 150.17,A -85,B 0,C 180,E1 -13811.83,E2 -13811.83} C_VEL
LIN {X 0,Y 347.706,Z 150.17,A -85,B 0,C 180,E1 -13815.026,E2 -13815.026} C_VEL
LIN {X 0,Y 347.751,Z 150.165,A -85,B 0,C 180,E1 -13818.397,E2 -13818.397} C_VEL
LIN {X 0,Y 347.773,Z 150.163,A -85,B 0,C 180,E1 -13822.011,E2 -13822.011} C_VEL
LIN {X 0,Y 347.744,Z 150.171,A -85,B 0,C 180,E1 -13825.536,E2 -13825.536} C_VEL
LIN {X 0,Y 347.764,Z 150.166,A -85,B 0,C 180,E1 -13829.653,E2 -13829.653} C_VEL
LIN {X 0,Y 347.852,Z 150.153,A -85,B 0,C 180,E1 -13832.744,E2 -13832.744} C_VEL
LIN {X 0,Y 347.786,Z 150.16,A -85,B 0,C 180,E1 -13836.161,E2 -13836.161} C_VEL
LIN {X 0,Y 347.8,Z 150.159,A -85,B 0,C 180,E1 -13839.908,E2 -13839.908} C_VEL
LIN {X 0,Y 347.832,Z 150.156,A -85,B 0,C 180,E1 -13843.568,E2 -13843.568} C_VEL
LIN {X 0,Y 347.89,Z 150.151,A -85,B 0,C 180,E1 -13847.16,E2 -13847.16} C_VEL
LIN {X 0,Y 347.935,Z 150.145,A -85,B 0,C 180,E1 -13850.7,E2 -13850.7} C_VEL
LIN {X 0,Y 348.05,Z 150.128,A -85,B 0,C 180,E1 -13854.205,E2 -13854.205} C_VEL
LIN {X 0,Y 348.206,Z 150.108,A -85,B 0,C 180,E1 -13857.686,E2 -13857.686} C_VEL
LIN {X 0,Y 348.344,Z 150.091,A -85,B 0,C 180,E1 -13860,E2 -13860} C_VEL
LIN {X 0,Y 348.207,Z 150.11,A -85,B 0,C 180,E1 -13862.313,E2 -13862.313} C_VEL
LIN {X 0,Y 348.09,Z 150.124,A -85,B 0,C 180,E1 -13866.958,E2 -13866.958} C_VEL
LIN {X 0,Y 347.928,Z 150.148,A -85,B 0,C 180,E1 -13870.474,E2 -13870.474} C_VEL
LIN {X 0,Y 347.898,Z 150.15,A -85,B 0,C 180,E1 -13874.15,E2 -13874.15} C_VEL
LIN {X 0,Y 347.89,Z 150.153,A -85,B 0,C 180,E1 -13878.29,E2 -13878.29} C_VEL
LIN {X 0,Y 347.767,Z 150.163,A -85,B 0,C 180,E1 -13881.626,E2 -13881.626} C_VEL
LIN {X 0,Y 347.81,Z 150.157,A -85,B 0,C 180,E1 -13885.108,E2 -13885.108} C_VEL
LIN {X 0,Y 347.807,Z 150.16,A -85,B 0,C 180,E1 -13887.694,E2 -13887.694} C_VEL
LIN {X 0,Y 347.748,Z 150.167,A -85,B 0,C 180,E1 -13890.348,E2 -13890.348} C_VEL
LIN {X 0,Y 347.747,Z 150.17,A -85,B 0,C 180,E1 -13894.044,E2 -13894.044} C_VEL
LIN {X 0,Y 347.761,Z 150.165,A -85,B 0,C 180,E1 -13897.321,E2 -13897.321} C_VEL
LIN {X 0,Y 347.731,Z 150.168,A -85,B 0,C 180,E1 -13900.297,E2 -13900.297} C_VEL
LIN {X 0,Y 347.722,Z 150.171,A -85,B 0,C 180,E1 -13903.408,E2 -13903.408} C_VEL
LIN {X 0,Y 347.724,Z 150.168,A -85,B 0,C 180,E1 -13906.686,E2 -13906.686} C_VEL
LIN {X 0,Y 347.746,Z 150.166,A -85,B 0,C 180,E1 -13910.173,E2 -13910.173} C_VEL
LIN {X 0,Y 347.76,Z 150.163,A -85,B 0,C 180,E1 -13912.679,E2 -13912.679} C_VEL
LIN {X 0,Y 347.747,Z 150.166,A -85,B 0,C 180,E1 -13915.956,E2 -13915.956} C_VEL
LIN {X 0,Y 347.763,Z 150.166,A -85,B 0,C 180,E1 -13919.654,E2 -13919.654} C_VEL
LIN {X 0,Y 347.851,Z 150.153,A -85,B 0,C 180,E1 -13922.745,E2 -13922.745} C_VEL
LIN {X 0,Y 347.785,Z 150.16,A -85,B 0,C 180,E1 -13926.162,E2 -13926.162} C_VEL
LIN {X 0,Y 347.799,Z 150.159,A -85,B 0,C 180,E1 -13929.909,E2 -13929.909} C_VEL
LIN {X 0,Y 347.832,Z 150.155,A -85,B 0,C 180,E1 -13933.569,E2 -13933.569} C_VEL
LIN {X 0,Y 347.889,Z 150.151,A -85,B 0,C 180,E1 -13937.161,E2 -13937.161} C_VEL
LIN {X 0,Y 347.935,Z 150.146,A -85,B 0,C 180,E1 -13940.701,E2 -13940.701} C_VEL
LIN {X 0,Y 348.05,Z 150.128,A -85,B 0,C 180,E1 -13944.206,E2 -13944.206} C_VEL
LIN {X 0,Y 347.976,Z 150.254,A -85,B 0,C 180,E1 -13946.599,E2 -13946.599} C_VEL
LIN {X 0,Y 349.123,Z 155.37,A -85,B 0,C 180,E1 -13948.035,E2 -13948.035} C_VEL
LIN {X 0,Y 353.568,Z 169.613,A -85,B 0,C 180,E1 -13948.583,E2 -13948.583} C_VEL
LIN {X 0,Y 355.567,Z 181.388,A -85,B 0,C 180,E1 -13948.94,E2 -13948.94} C_VEL
LIN {X 0,Y 353.994,Z 262.308,A -85,B 0,C 180,E1 -13950.605,E2 -13950.605} C_VEL
LIN {X 0,Y 353.517,Z 275.625,A -85,B 0,C 180,E1 -13951.104,E2 -13951.104} C_VEL
LIN {X 0,Y 352.929,Z 288.907,A -85,B 0,C 180,E1 -13951.855,E2 -13951.855} C_VEL
LIN {X 0,Y 352.108,Z 301.192,A -85,B 0,C 180,E1 -13952.811,E2 -13952.811} C_VEL
LIN {X 0,Y 351.15,Z 313.123,A -85,B 0,C 180,E1 -13954.017,E2 -13954.017} C_VEL
LIN {X 0,Y 350.162,Z 323.381,A -85,B 0,C 180,E1 -13955.326,E2 -13955.326} C_VEL
LIN {X 0,Y 349.087,Z 333.463,A -85,B 0,C 180,E1 -13956.938,E2 -13956.938} C_VEL
LIN {X 0,Y 348.291,Z 341.831,A -85,B 0,C 180,E1 -13958.605,E2 -13958.605} C_VEL
LIN {X 0,Y 347.53,Z 349.311,A -85,B 0,C 180,E1 -13960.487,E2 -13960.487} C_VEL
LIN {X 0,Y 347.025,Z 354.926,A -85,B 0,C 180,E1 -13962.278,E2 -13962.278} C_VEL
LIN {X 0,Y 346.632,Z 359.319,A -85,B 0,C 180,E1 -13964.082,E2 -13964.082} C_VEL
LIN {X 0,Y 346.407,Z 361.651,A -85,B 0,C 180,E1 -13965.293,E2 -13965.293} C_VEL
LIN {X 0,Y 346.185,Z 364.526,A -85,B 0,C 180,E1 -13967.416,E2 -13967.416} C_VEL
LIN {X 0,Y 346.103,Z 365.79,A -85,B 0,C 180,E1 -13968.96,E2 -13968.96} C_VEL
LIN {X 0,Y 346.143,Z 366.361,A -85,B 0,C 180,E1 -13970.938,E2 -13970.938} C_VEL
LIN {X 0,Y 346.242,Z 365.924,A -85,B 0,C 180,E1 -13972.685,E2 -13972.685} C_VEL
LIN {X 0,Y 346.438,Z 364.902,A -85,B 0,C 180,E1 -13974.093,E2 -13974.093} C_VEL
LIN {X 0,Y 346.632,Z 363.705,A -85,B 0,C 180,E1 -13975.2,E2 -13975.2} C_VEL
LIN {X 0,Y 347.094,Z 360.927,A -85,B 0,C 180,E1 -13977.012,E2 -13977.012} C_VEL
LIN {X 0,Y 347.777,Z 356.613,A -85,B 0,C 180,E1 -13979.013,E2 -13979.013} C_VEL
LIN {X 0,Y 348.632,Z 351.051,A -85,B 0,C 180,E1 -13980.934,E2 -13980.934} C_VEL
LIN {X 0,Y 349.783,Z 343.853,A -85,B 0,C 180,E1 -13982.854,E2 -13982.854} C_VEL
LIN {X 0,Y 350.392,Z 339.816,A -85,B 0,C 180,E1 -13983.76,E2 -13983.76} C_VEL
LIN {X 0,Y 350.29,Z 336.251,A -85,B 0,C 180,E1 -13984.532,E2 -13984.532} C_VEL
LIN {X 0,Y 348.45,Z 330.218,A -85,B 0,C 180,E1 -13985.791,E2 -13985.791} C_VEL
LIN {X 0,Y 346.736,Z 323.665,A -85,B 0,C 180,E1 -13986.976,E2 -13986.976} C_VEL
LIN {X 0,Y 346.812,Z 319.224,A -85,B 0,C 180,E1 -13987.62,E2 -13987.62} C_VEL
LIN {X 0,Y 348.292,Z 308.113,A -85,B 0,C 180,E1 -13988.907,E2 -13988.907} C_VEL
LIN {X 0,Y 349.691,Z 295.745,A -85,B 0,C 180,E1 -13990.026,E2 -13990.026} C_VEL
LIN {X 0,Y 350.649,Z 283.436,A -85,B 0,C 180,E1 -13990.865,E2 -13990.865} C_VEL
LIN {X 0,Y 351.448,Z 270.611,A -85,B 0,C 180,E1 -13991.481,E2 -13991.481} C_VEL
LIN {X 0,Y 351.937,Z 257.236,A -85,B 0,C 180,E1 -13991.881,E2 -13991.881} C_VEL
LIN {X 0,Y 353.702,Z 183.674,A -85,B 0,C 180,E1 -13993.428,E2 -13993.428} C_VEL
LIN {X 0,Y 351.584,Z 177.802,A -85,B 0,C 180,E1 -13993.75,E2 -13993.75} C_VEL
LIN {X 0,Y 344.786,Z 162.505,A -85,B 0,C 180,E1 -13994.731,E2 -13994.731} C_VEL
LIN {X 0,Y 342.059,Z 156.64,A -85,B 0,C 180,E1 -13995.171,E2 -13995.171} C_VEL
LIN {X 0,Y 340.662,Z 151.052,A -85,B 0,C 180,E1 -13996.995,E2 -13996.995} C_VEL
LIN {X 0,Y 340.655,Z 151.046,A -85,B 0,C 180,E1 -14000.242,E2 -14000.242} C_VEL
LIN {X 0,Y 340.707,Z 151.035,A -85,B 0,C 180,E1 -14003.56,E2 -14003.56} C_VEL
LIN {X 0,Y 340.692,Z 151.046,A -85,B 0,C 180,E1 -14006.154,E2 -14006.154} C_VEL
LIN {X 0,Y 340.721,Z 151.046,A -85,B 0,C 180,E1 -14010.035,E2 -14010.035} C_VEL
LIN {X 0,Y 340.71,Z 151.048,A -85,B 0,C 180,E1 -14013.012,E2 -14013.012} C_VEL
LIN {X 0,Y 340.697,Z 151.042,A -85,B 0,C 180,E1 -14016.925,E2 -14016.925} C_VEL
LIN {X 0,Y 340.697,Z 151.04,A -85,B 0,C 180,E1 -14020.728,E2 -14020.728} C_VEL
LIN {X 0,Y 340.726,Z 151.042,A -85,B 0,C 180,E1 -14023.216,E2 -14023.216} C_VEL
LIN {X 0,Y 340.815,Z 151.031,A -85,B 0,C 180,E1 -14026.89,E2 -14026.89} C_VEL
LIN {X 0,Y 340.88,Z 151.023,A -85,B 0,C 180,E1 -14030.507,E2 -14030.507} C_VEL
LIN {X 0,Y 341.003,Z 150.999,A -85,B 0,C 180,E1 -14032.897,E2 -14032.897} C_VEL
LIN {X 0,Y 340.807,Z 151.029,A -85,B 0,C 180,E1 -14035.269,E2 -14035.269} C_VEL
LIN {X 0,Y 341.118,Z 150.985,A -85,B 0,C 180,E1 -14037.639,E2 -14037.639} C_VEL
LIN {X 0,Y 341.089,Z 150.995,A -85,B 0,C 180,E1 -14041.181,E2 -14041.181} C_VEL
LIN {X 0,Y 341.125,Z 150.981,A -85,B 0,C 180,E1 -14042.362,E2 -14042.362} C_VEL
LIN {X 0,Y 341.016,Z 151.005,A -85,B 0,C 180,E1 -14045.915,E2 -14045.915} C_VEL
LIN {X 0,Y 340.965,Z 151.004,A -85,B 0,C 180,E1 -14048.356,E2 -14048.356} C_VEL
LIN {X 0,Y 340.851,Z 151.019,A -85,B 0,C 180,E1 -14051.899,E2 -14051.899} C_VEL
LIN {X 0,Y 340.819,Z 151.031,A -85,B 0,C 180,E1 -14055.55,E2 -14055.55} C_VEL
LIN {X 0,Y 340.765,Z 151.035,A -85,B 0,C 180,E1 -14059.268,E2 -14059.268} C_VEL
LIN {X 0,Y 340.72,Z 151.035,A -85,B 0,C 180,E1 -14063.074,E2 -14063.074} C_VEL
LIN {X 0,Y 340.722,Z 151.036,A -85,B 0,C 180,E1 -14065.669,E2 -14065.669} C_VEL
LIN {X 0,Y 340.71,Z 151.039,A -85,B 0,C 180,E1 -14069.674,E2 -14069.674} C_VEL
LIN {X 0,Y 340.688,Z 151.048,A -85,B 0,C 180,E1 -14072.436,E2 -14072.436} C_VEL
LIN {X 0,Y 340.72,Z 151.044,A -85,B 0,C 180,E1 -14075.279,E2 -14075.279} C_VEL
LIN {X 0,Y 340.696,Z 151.045,A -85,B 0,C 180,E1 -14078.383,E2 -14078.383} C_VEL
LIN {X 0,Y 340.696,Z 151.049,A -85,B 0,C 180,E1 -14082.044,E2 -14082.044} C_VEL
LIN {X 0,Y 340.654,Z 151.053,A -85,B 0,C 180,E1 -14086.227,E2 -14086.227} C_VEL
LIN {X 0,Y 340.689,Z 151.049,A -85,B 0,C 180,E1 -14089.753,E2 -14089.753} C_VEL
LIN {X 0,Y 340.707,Z 151.04,A -85,B 0,C 180,E1 -14093.258,E2 -14093.258} C_VEL
LIN {X 0,Y 340.716,Z 151.116,A -85,B 0,C 180,E1 -14096.422,E2 -14096.422} C_VEL
LIN {X 0,Y 343.415,Z 161.856,A -85,B 0,C 180,E1 -14099.599,E2 -14099.599} C_VEL
LIN {X 0,Y 345.414,Z 170.84,A -85,B 0,C 180,E1 -14102.097,E2 -14102.097} C_VEL
LIN {X 0,Y 346.247,Z 176.067,A -85,B 0,C 180,E1 -14103.477,E2 -14103.477} C_VEL
LIN {X 0,Y 345.411,Z 183.57,A -85,B 0,C 180,E1 -14105.243,E2 -14105.243} C_VEL
LIN {X 0,Y 350.618,Z 209.569,A -85,B 0,C 180,E1 -14106.319,E2 -14106.319} C_VEL
LIN {X 0,Y 352.818,Z 225.168,A -85,B 0,C 180,E1 -14106.867,E2 -14106.867} C_VEL
LIN {X 0,Y 351.207,Z 292.54,A -85,B 0,C 180,E1 -14108.31,E2 -14108.31} C_VEL
LIN {X 0,Y 350.305,Z 305.65,A -85,B 0,C 180,E1 -14108.792,E2 -14108.792} C_VEL
LIN {X 0,Y 349.06,Z 318.862,A -85,B 0,C 180,E1 -14109.523,E2 -14109.523} C_VEL
LIN {X 0,Y 347.808,Z 330.003,A -85,B 0,C 180,E1 -14110.37,E2 -14110.37} C_VEL
LIN {X 0,Y 346.307,Z 341.586,A -85,B 0,C 180,E1 -14111.512,E2 -14111.512} C_VEL
LIN {X 0,Y 344.779,Z 352.04,A -85,B 0,C 180,E1 -14112.808,E2 -14112.808} C_VEL
LIN {X 0,Y 343.478,Z 360.443,A -85,B 0,C 180,E1 -14114.088,E2 -14114.088} C_VEL
LIN {X 0,Y 342.247,Z 369.264,A -85,B 0,C 180,E1 -14115.734,E2 -14115.734} C_VEL
LIN {X 0,Y 341.013,Z 376.89,A -85,B 0,C 180,E1 -14117.502,E2 -14117.502} C_VEL
LIN {X 0,Y 340.17,Z 383.054,A -85,B 0,C 180,E1 -14119.284,E2 -14119.284} C_VEL
LIN {X 0,Y 339.588,Z 387.971,A -85,B 0,C 180,E1 -14121.07,E2 -14121.07} C_VEL
LIN {X 0,Y 339.251,Z 391.78,A -85,B 0,C 180,E1 -14122.86,E2 -14122.86} C_VEL
LIN {X 0,Y 339.13,Z 393.864,A -85,B 0,C 180,E1 -14124.121,E2 -14124.121} C_VEL
LIN {X 0,Y 339.072,Z 395.325,A -85,B 0,C 180,E1 -14125.244,E2 -14125.244} C_VEL
LIN {X 0,Y 339.088,Z 396.443,A -85,B 0,C 180,E1 -14126.435,E2 -14126.435} C_VEL
LIN {X 0,Y 339.161,Z 397.494,A -85,B 0,C 180,E1 -14128.812,E2 -14128.812} C_VEL
LIN {X 0,Y 339.228,Z 397.438,A -85,B 0,C 180,E1 -14130,E2 -14130} C_VEL
LIN {X 0,Y 339.188,Z 396.943,A -85,B 0,C 180,E1 -14131.187,E2 -14131.187} C_VEL
LIN {X 0,Y 339.105,Z 394.725,A -85,B 0,C 180,E1 -14133.564,E2 -14133.564} C_VEL
LIN {X 0,Y 339.079,Z 391.851,A -85,B 0,C 180,E1 -14135.394,E2 -14135.394} C_VEL
LIN {X 0,Y 339.231,Z 388.087,A -85,B 0,C 180,E1 -14137.14,E2 -14137.14} C_VEL
LIN {X 0,Y 339.496,Z 383.091,A -85,B 0,C 180,E1 -14138.932,E2 -14138.932} C_VEL
LIN {X 0,Y 339.927,Z 376.789,A -85,B 0,C 180,E1 -14140.724,E2 -14140.724} C_VEL
LIN {X 0,Y 340.75,Z 368.91,A -85,B 0,C 180,E1 -14142.507,E2 -14142.507} C_VEL
LIN {X 0,Y 341.56,Z 360.84,A -85,B 0,C 180,E1 -14143.991,E2 -14143.991} C_VEL
LIN {X 0,Y 342.418,Z 350.965,A -85,B 0,C 180,E1 -14145.475,E2 -14145.475} C_VEL
LIN {X 0,Y 343.569,Z 339.993,A -85,B 0,C 180,E1 -14146.794,E2 -14146.794} C_VEL
LIN {X 0,Y 344.506,Z 329.221,A -85,B 0,C 180,E1 -14147.818,E2 -14147.818} C_VEL
LIN {X 0,Y 345.608,Z 316.279,A -85,B 0,C 180,E1 -14148.756,E2 -14148.756} C_VEL
LIN {X 0,Y 346.486,Z 303.122,A -85,B 0,C 180,E1 -14149.437,E2 -14149.437} C_VEL
LIN {X 0,Y 347.018,Z 289.988,A -85,B 0,C 180,E1 -14149.868,E2 -14149.868} C_VEL
LIN {X 0,Y 348.056,Z 222.158,A -85,B 0,C 180,E1 -14151.295,E2 -14151.295} C_VEL
LIN {X 0,Y 342.958,Z 184.587,A -85,B 0,C 180,E1 -14152.398,E2 -14152.398} C_VEL
LIN {X 0,Y 344.288,Z 171.478,A -85,B 0,C 180,E1 -14155.383,E2 -14155.383} C_VEL
LIN {X 0,Y 344.096,Z 167.576,A -85,B 0,C 180,E1 -14156.31,E2 -14156.31} C_VEL
LIN {X 0,Y 341.798,Z 155.956,A -85,B 0,C 180,E1 -14159.232,E2 -14159.232} C_VEL
LIN {X 0,Y 340.736,Z 151.044,A -85,B 0,C 180,E1 -14160.555,E2 -14160.555} C_VEL
LIN {X 0,Y 340.724,Z 151.042,A -85,B 0,C 180,E1 -14164.404,E2 -14164.404} C_VEL
LIN {X 0,Y 340.711,Z 151.043,A -85,B 0,C 180,E1 -14168.386,E2 -14168.386} C_VEL
LIN {X 0,Y 340.7,Z 151.046,A -85,B 0,C 180,E1 -14172.045,E2 -14172.045} C_VEL
LIN {X 0,Y 340.652,Z 151.05,A -85,B 0,C 180,E1 -14176.227,E2 -14176.227} C_VEL
LIN {X 0,Y 340.689,Z 151.049,A -85,B 0,C 180,E1 -14179.753,E2 -14179.753} C_VEL
LIN {X 0,Y 340.705,Z 151.045,A -85,B 0,C 180,E1 -14183.258,E2 -14183.258} C_VEL
LIN {X 0,Y 340.692,Z 151.044,A -85,B 0,C 180,E1 -14186.153,E2 -14186.153} C_VEL
LIN {X 0,Y 340.775,Z 151.033,A -85,B 0,C 180,E1 -14190.332,E2 -14190.332} C_VEL
LIN {X 0,Y 340.805,Z 151.033,A -85,B 0,C 180,E1 -14193.02,E2 -14193.02} C_VEL
LIN {X 0,Y 340.755,Z 151.038,A -85,B 0,C 180,E1 -14195.638,E2 -14195.638} C_VEL
LIN {X 0,Y 340.73,Z 151.042,A -85,B 0,C 180,E1 -14199.473,E2 -14199.473} C_VEL
LIN {X 0,Y 340.792,Z 151.031,A -85,B 0,C 180,E1 -14201.98,E2 -14201.98} C_VEL
LIN {X 0,Y 340.869,Z 151.022,A -85,B 0,C 180,E1 -14205.705,E2 -14205.705} C_VEL
LIN {X 0,Y 340.848,Z 151.027,A -85,B 0,C 180,E1 -14209.305,E2 -14209.305} C_VEL
LIN {X 0,Y 341.009,Z 151.01,A -85,B 0,C 180,E1 -14212.897,E2 -14212.897} C_VEL
LIN {X 0,Y 341.168,Z 150.984,A -85,B 0,C 180,E1 -14217.639,E2 -14217.639} C_VEL
LIN {X 0,Y 341.295,Z 150.969,A -85,B 0,C 180,E1 -14220,E2 -14220} C_VEL
LIN {X 0,Y 341.169,Z 150.988,A -85,B 0,C 180,E1 -14222.361,E2 -14222.361} C_VEL
LIN {X 0,Y 341.058,Z 150.999,A -85,B 0,C 180,E1 -14227.102,E2 -14227.102} C_VEL
LIN {X 0,Y 340.87,Z 151.025,A -85,B 0,C 180,E1 -14230.694,E2 -14230.694} C_VEL
LIN {X 0,Y 340.862,Z 151.028,A -85,B 0,C 180,E1 -14234.325,E2 -14234.325} C_VEL
LIN {X 0,Y 340.836,Z 151.03,A -85,B 0,C 180,E1 -14238.466,E2 -14238.466} C_VEL
LIN {X 0,Y 340.716,Z 151.043,A -85,B 0,C 180,E1 -14241.842,E2 -14241.842} C_VEL
LIN {X 0,Y 340.771,Z 151.036,A -85,B 0,C 180,E1 -14245.664,E2 -14245.664} C_VEL
LIN {X 0,Y 340.727,Z 151.042,A -85,B 0,C 180,E1 -14248.321,E2 -14248.321} C_VEL
LIN {X 0,Y 340.697,Z 151.043,A -85,B 0,C 180,E1 -14251.045,E2 -14251.045} C_VEL
LIN {X 0,Y 340.717,Z 151.042,A -85,B 0,C 180,E1 -14255.279,E2 -14255.279} C_VEL
LIN {X 0,Y 340.708,Z 151.043,A -85,B 0,C 180,E1 -14258.386,E2 -14258.386} C_VEL
LIN {X 0,Y 340.698,Z 151.046,A -85,B 0,C 180,E1 -14262.045,E2 -14262.045} C_VEL
LIN {X 0,Y 340.65,Z 151.05,A -85,B 0,C 180,E1 -14266.227,E2 -14266.227} C_VEL
LIN {X 0,Y 340.687,Z 151.048,A -85,B 0,C 180,E1 -14269.753,E2 -14269.753} C_VEL
LIN {X 0,Y 340.703,Z 151.046,A -85,B 0,C 180,E1 -14273.259,E2 -14273.259} C_VEL
LIN {X 0,Y 340.691,Z 151.044,A -85,B 0,C 180,E1 -14276.153,E2 -14276.153} C_VEL
LIN {X 0,Y 340.774,Z 151.033,A -85,B 0,C 180,E1 -14280.333,E2 -14280.333} C_VEL
LIN {X 0,Y 340.804,Z 151.033,A -85,B 0,C 180,E1 -14283.02,E2 -14283.02} C_VEL
LIN {X 0,Y 340.754,Z 151.038,A -85,B 0,C 180,E1 -14285.638,E2 -14285.638} C_VEL
LIN {X 0,Y 340.729,Z 151.041,A -85,B 0,C 180,E1 -14289.473,E2 -14289.473} C_VEL
LIN {X 0,Y 340.791,Z 151.031,A -85,B 0,C 180,E1 -14291.981,E2 -14291.981} C_VEL
LIN {X 0,Y 340.869,Z 151.022,A -85,B 0,C 180,E1 -14295.705,E2 -14295.705} C_VEL
LIN {X 0,Y 340.848,Z 151.026,A -85,B 0,C 180,E1 -14299.306,E2 -14299.306} C_VEL
LIN {X 0,Y 341.009,Z 151.009,A -85,B 0,C 180,E1 -14302.897,E2 -14302.897} C_VEL
LIN {X 0,Y 340.916,Z 151.151,A -85,B 0,C 180,E1 -14306.344,E2 -14306.344} C_VEL
LIN {X 0,Y 342.021,Z 155.677,A -85,B 0,C 180,E1 -14307.645,E2 -14307.645} C_VEL
LIN {X 0,Y 346.945,Z 171.247,A -85,B 0,C 180,E1 -14308.264,E2 -14308.264} C_VEL
LIN {X 0,Y 348.791,Z 182.34,A -85,B 0,C 180,E1 -14308.607,E2 -14308.607} C_VEL
LIN {X 0,Y 347.152,Z 263.733,A -85,B 0,C 180,E1 -14310.326,E2 -14310.326} C_VEL
LIN {X 0,Y 346.658,Z 277.409,A -85,B 0,C 180,E1 -14310.871,E2 -14310.871} C_VEL
LIN {X 0,Y 346.047,Z 289.74,A -85,B 0,C 180,E1 -14311.6,E2 -14311.6} C_VEL
LIN {X 0,Y 345.167,Z 302.175,A -85,B 0,C 180,E1 -14312.601,E2 -14312.601} C_VEL
LIN {X 0,Y 344.19,Z 313.767,A -85,B 0,C 180,E1 -14313.805,E2 -14313.805} C_VEL
LIN {X 0,Y 343.266,Z 322.941,A -85,B 0,C 180,E1 -14314.992,E2 -14314.992} C_VEL
LIN {X 0,Y 342.279,Z 332.319,A -85,B 0,C 180,E1 -14316.485,E2 -14316.485} C_VEL
LIN {X 0,Y 341.355,Z 341.411,A -85,B 0,C 180,E1 -14318.287,E2 -14318.287} C_VEL
LIN {X 0,Y 340.584,Z 348.722,A -85,B 0,C 180,E1 -14320.102,E2 -14320.102} C_VEL
LIN {X 0,Y 340.005,Z 354.523,A -85,B 0,C 180,E1 -14321.929,E2 -14321.929} C_VEL
LIN {X 0,Y 339.677,Z 358.471,A -85,B 0,C 180,E1 -14323.483,E2 -14323.483} C_VEL
LIN {X 0,Y 339.249,Z 362.517,A -85,B 0,C 180,E1 -14325.624,E2 -14325.624} C_VEL
LIN {X 0,Y 339.089,Z 364.966,A -85,B 0,C 180,E1 -14327.561,E2 -14327.561} C_VEL
LIN {X 0,Y 338.993,Z 366.279,A -85,B 0,C 180,E1 -14329.373,E2 -14329.373} C_VEL
LIN {X 0,Y 339.062,Z 366.678,A -85,B 0,C 180,E1 -14331.133,E2 -14331.133} C_VEL
LIN {X 0,Y 339.208,Z 366.037,A -85,B 0,C 180,E1 -14333.183,E2 -14333.183} C_VEL
LIN {X 0,Y 339.421,Z 365.041,A -85,B 0,C 180,E1 -14334.464,E2 -14334.464} C_VEL
LIN {X 0,Y 339.855,Z 362.648,A -85,B 0,C 180,E1 -14336.398,E2 -14336.398} C_VEL
LIN {X 0,Y 340.469,Z 359.092,A -85,B 0,C 180,E1 -14338.344,E2 -14338.344} C_VEL
LIN {X 0,Y 341.317,Z 353.77,A -85,B 0,C 180,E1 -14340.457,E2 -14340.457} C_VEL
LIN {X 0,Y 342.336,Z 347.833,A -85,B 0,C 180,E1 -14342.261,E2 -14342.261} C_VEL
LIN {X 0,Y 343.658,Z 339.676,A -85,B 0,C 180,E1 -14344.221,E2 -14344.221} C_VEL
LIN {X 0,Y 345.122,Z 330.753,A -85,B 0,C 180,E1 -14345.903,E2 -14345.903} C_VEL
LIN {X 0,Y 346.469,Z 321.594,A -85,B 0,C 180,E1 -14347.301,E2 -14347.301} C_VEL
LIN {X 0,Y 346.812,Z 319.224,A -85,B 0,C 180,E1 -14347.62,E2 -14347.62} C_VEL
LIN {X 0,Y 346.898,Z 314.646,A -85,B 0,C 180,E1 -14348.24,E2 -14348.24} C_VEL
LIN {X 0,Y 345.241,Z 307.107,A -85,B 0,C 180,E1 -14349.276,E2 -14349.276} C_VEL
LIN {X 0,Y 343.483,Z 299.163,A -85,B 0,C 180,E1 -14350.218,E2 -14350.218} C_VEL
LIN {X 0,Y 343.39,Z 293.952,A -85,B 0,C 180,E1 -14350.68,E2 -14350.68} C_VEL
LIN {X 0,Y 344.469,Z 280.813,A -85,B 0,C 180,E1 -14351.535,E2 -14351.535} C_VEL
LIN {X 0,Y 345.241,Z 267.921,A -85,B 0,C 180,E1 -14352.106,E2 -14352.106} C_VEL
LIN {X 0,Y 345.715,Z 252.761,A -85,B 0,C 180,E1 -14352.502,E2 -14352.502} C_VEL
LIN {X 0,Y 347.453,Z 184.995,A -85,B 0,C 180,E1 -14353.949,E2 -14353.949} C_VEL
LIN {X 0,Y 339.764,Z 167.052,A -85,B 0,C 180,E1 -14355.099,E2 -14355.099} C_VEL
LIN {X 0,Y 334.922,Z 157.121,A -85,B 0,C 180,E1 -14355.84,E2 -14355.84} C_VEL
LIN {X 0,Y 333.635,Z 151.926,A -85,B 0,C 180,E1 -14357.618,E2 -14357.618} C_VEL
LIN {X 0,Y 333.616,Z 151.927,A -85,B 0,C 180,E1 -14361.21,E2 -14361.21} C_VEL
LIN {X 0,Y 333.673,Z 151.911,A -85,B 0,C 180,E1 -14363.861,E2 -14363.861} C_VEL
LIN {X 0,Y 333.644,Z 151.928,A -85,B 0,C 180,E1 -14367.414,E2 -14367.414} C_VEL
LIN {X 0,Y 333.631,Z 151.926,A -85,B 0,C 180,E1 -14371.021,E2 -14371.021} C_VEL
LIN {X 0,Y 333.658,Z 151.923,A -85,B 0,C 180,E1 -14374.922,E2 -14374.922} C_VEL
LIN {X 0,Y 333.641,Z 151.927,A -85,B 0,C 180,E1 -14379.017,E2 -14379.017} C_VEL
LIN {X 0,Y 333.706,Z 151.911,A -85,B 0,C 180,E1 -14381.585,E2 -14381.585} C_VEL
LIN {X 0,Y 333.759,Z 151.904,A -85,B 0,C 180,E1 -14385.611,E2 -14385.611} C_VEL
LIN {X 0,Y 333.809,Z 151.893,A -85,B 0,C 180,E1 -14389.077,E2 -14389.077} C_VEL
LIN {X 0,Y 333.958,Z 151.877,A -85,B 0,C 180,E1 -14392.746,E2 -14392.746} C_VEL
LIN {X 0,Y 333.774,Z 151.904,A -85,B 0,C 180,E1 -14395.169,E2 -14395.169} C_VEL
LIN {X 0,Y 334.058,Z 151.864,A -85,B 0,C 180,E1 -14397.589,E2 -14397.589} C_VEL
LIN {X 0,Y 334.059,Z 151.871,A -85,B 0,C 180,E1 -14401.206,E2 -14401.206} C_VEL
LIN {X 0,Y 334.066,Z 151.86,A -85,B 0,C 180,E1 -14402.412,E2 -14402.412} C_VEL
LIN {X 0,Y 333.989,Z 151.879,A -85,B 0,C 180,E1 -14406.04,E2 -14406.04} C_VEL
LIN {X 0,Y 333.822,Z 151.902,A -85,B 0,C 180,E1 -14409.697,E2 -14409.697} C_VEL
LIN {X 0,Y 333.799,Z 151.895,A -85,B 0,C 180,E1 -14413.392,E2 -14413.392} C_VEL
LIN {X 0,Y 333.721,Z 151.907,A -85,B 0,C 180,E1 -14417.148,E2 -14417.148} C_VEL
LIN {X 0,Y 333.72,Z 151.915,A -85,B 0,C 180,E1 -14419.692,E2 -14419.692} C_VEL
LIN {X 0,Y 333.665,Z 151.92,A -85,B 0,C 180,E1 -14423.591,E2 -14423.591} C_VEL
LIN {X 0,Y 333.659,Z 151.914,A -85,B 0,C 180,E1 -14426.253,E2 -14426.253} C_VEL
LIN {X 0,Y 333.664,Z 151.916,A -85,B 0,C 180,E1 -14430.278,E2 -14430.278} C_VEL
LIN {X 0,Y 333.639,Z 151.922,A -85,B 0,C 180,E1 -14433.208,E2 -14433.208} C_VEL
LIN {X 0,Y 333.677,Z 151.921,A -85,B 0,C 180,E1 -14436.139,E2 -14436.139} C_VEL
LIN {X 0,Y 333.622,Z 151.928,A -85,B 0,C 180,E1 -14439.196,E2 -14439.196} C_VEL
LIN {X 0,Y 333.631,Z 151.928,A -85,B 0,C 180,E1 -14442.499,E2 -14442.499} C_VEL
LIN {X 0,Y 333.598,Z 151.931,A -85,B 0,C 180,E1 -14445.955,E2 -14445.955} C_VEL
LIN {X 0,Y 333.649,Z 151.927,A -85,B 0,C 180,E1 -14449.315,E2 -14449.315} C_VEL
LIN {X 0,Y 333.667,Z 151.916,A -85,B 0,C 180,E1 -14453.168,E2 -14453.168} C_VEL
LIN {X 0,Y 333.672,Z 151.94,A -85,B 0,C 180,E1 -14455.798,E2 -14455.798} C_VEL
LIN {X 0,Y 335.876,Z 160.623,A -85,B 0,C 180,E1 -14458.459,E2 -14458.459} C_VEL
LIN {X 0,Y 338.276,Z 170.944,A -85,B 0,C 180,E1 -14461.455,E2 -14461.455} C_VEL
LIN {X 0,Y 339.404,Z 177.325,A -85,B 0,C 180,E1 -14463.196,E2 -14463.196} C_VEL
LIN {X 0,Y 338.795,Z 183.269,A -85,B 0,C 180,E1 -14464.616,E2 -14464.616} C_VEL
LIN {X 0,Y 344.067,Z 208.991,A -85,B 0,C 180,E1 -14465.728,E2 -14465.728} C_VEL
LIN {X 0,Y 346.485,Z 225.358,A -85,B 0,C 180,E1 -14466.331,E2 -14466.331} C_VEL
LIN {X 0,Y 344.804,Z 292.756,A -85,B 0,C 180,E1 -14467.808,E2 -14467.808} C_VEL
LIN {X 0,Y 343.821,Z 306.41,A -85,B 0,C 180,E1 -14468.333,E2 -14468.333} C_VEL
LIN {X 0,Y 342.586,Z 318.751,A -85,B 0,C 180,E1 -14469.039,E2 -14469.039} C_VEL
LIN {X 0,Y 341.171,Z 330.595,A -85,B 0,C 180,E1 -14469.972,E2 -14469.972} C_VEL
LIN {X 0,Y 339.615,Z 341.987,A -85,B 0,C 180,E1 -14471.135,E2 -14471.135} C_VEL
LIN {X 0,Y 337.994,Z 352.296,A -85,B 0,C 180,E1 -14472.452,E2 -14472.452} C_VEL
LIN {X 0,Y 336.392,Z 362.207,A -85,B 0,C 180,E1 -14474.045,E2 -14474.045} C_VEL
LIN {X 0,Y 335.154,Z 370.656,A -85,B 0,C 180,E1 -14475.736,E2 -14475.736} C_VEL
LIN {X 0,Y 333.87,Z 377.982,A -85,B 0,C 180,E1 -14477.539,E2 -14477.539} C_VEL
LIN {X 0,Y 332.914,Z 384.728,A -85,B 0,C 180,E1 -14479.663,E2 -14479.663} C_VEL
LIN {X 0,Y 332.411,Z 389.213,A -85,B 0,C 180,E1 -14481.489,E2 -14481.489} C_VEL
LIN {X 0,Y 332.178,Z 391.594,A -85,B 0,C 180,E1 -14482.707,E2 -14482.707} C_VEL
LIN {X 0,Y 332.029,Z 393.916,A -85,B 0,C 180,E1 -14484.181,E2 -14484.181} C_VEL
LIN {X 0,Y 332.011,Z 396.17,A -85,B 0,C 180,E1 -14486.359,E2 -14486.359} C_VEL
LIN {X 0,Y 332.063,Z 397.179,A -85,B 0,C 180,E1 -14488.787,E2 -14488.787} C_VEL
LIN {X 0,Y 332.136,Z 397.093,A -85,B 0,C 180,E1 -14490,E2 -14490} C_VEL
LIN {X 0,Y 332.091,Z 396.563,A -85,B 0,C 180,E1 -14491.212,E2 -14491.212} C_VEL
LIN {X 0,Y 332.03,Z 394.302,A -85,B 0,C 180,E1 -14493.641,E2 -14493.641} C_VEL
LIN {X 0,Y 332.027,Z 390.813,A -85,B 0,C 180,E1 -14495.816,E2 -14495.816} C_VEL
LIN {X 0,Y 332.243,Z 386.013,A -85,B 0,C 180,E1 -14497.903,E2 -14497.903} C_VEL
LIN {X 0,Y 332.659,Z 379.513,A -85,B 0,C 180,E1 -14500.037,E2 -14500.037} C_VEL
LIN {X 0,Y 333.314,Z 372.388,A -85,B 0,C 180,E1 -14501.863,E2 -14501.863} C_VEL
LIN {X 0,Y 334.204,Z 363.462,A -85,B 0,C 180,E1 -14503.684,E2 -14503.684} C_VEL
LIN {X 0,Y 334.996,Z 355.359,A -85,B 0,C 180,E1 -14505.036,E2 -14505.036} C_VEL
LIN {X 0,Y 336.039,Z 345.398,A -85,B 0,C 180,E1 -14506.4,E2 -14506.4} C_VEL
LIN {X 0,Y 337.097,Z 334.512,A -85,B 0,C 180,E1 -14507.596,E2 -14507.596} C_VEL
LIN {X 0,Y 338.243,Z 322.298,A -85,B 0,C 180,E1 -14508.63,E2 -14508.63} C_VEL
LIN {X 0,Y 339.229,Z 309.537,A -85,B 0,C 180,E1 -14509.437,E2 -14509.437} C_VEL
LIN {X 0,Y 339.937,Z 296.903,A -85,B 0,C 180,E1 -14509.985,E2 -14509.985} C_VEL
LIN {X 0,Y 340.434,Z 279.166,A -85,B 0,C 180,E1 -14510.427,E2 -14510.427} C_VEL
LIN {X 0,Y 341.29,Z 222.943,A -85,B 0,C 180,E1 -14511.627,E2 -14511.627} C_VEL
LIN {X 0,Y 336.073,Z 184.2,A -85,B 0,C 180,E1 -14512.801,E2 -14512.801} C_VEL
LIN {X 0,Y 337.332,Z 172.12,A -85,B 0,C 180,E1 -14515.614,E2 -14515.614} C_VEL
LIN {X 0,Y 336.878,Z 167.491,A -85,B 0,C 180,E1 -14516.752,E2 -14516.752} C_VEL
LIN {X 0,Y 334.385,Z 155.122,A -85,B 0,C 180,E1 -14519.945,E2 -14519.945} C_VEL
LIN {X 0,Y 333.705,Z 151.92,A -85,B 0,C 180,E1 -14520.798,E2 -14520.798} C_VEL
LIN {X 0,Y 333.687,Z 151.917,A -85,B 0,C 180,E1 -14524.774,E2 -14524.774} C_VEL
LIN {X 0,Y 333.653,Z 151.925,A -85,B 0,C 180,E1 -14527.651,E2 -14527.651} C_VEL
LIN {X 0,Y 333.647,Z 151.921,A -85,B 0,C 180,E1 -14530.767,E2 -14530.767} C_VEL
LIN {X 0,Y 333.594,Z 151.929,A -85,B 0,C 180,E1 -14534.25,E2 -14534.25} C_VEL
LIN {X 0,Y 333.642,Z 151.928,A -85,B 0,C 180,E1 -14537.618,E2 -14537.618} C_VEL
LIN {X 0,Y 333.653,Z 151.923,A -85,B 0,C 180,E1 -14541.202,E2 -14541.202} C_VEL
LIN {X 0,Y 333.676,Z 151.92,A -85,B 0,C 180,E1 -14543.861,E2 -14543.861} C_VEL
LIN {X 0,Y 333.643,Z 151.928,A -85,B 0,C 180,E1 -14547.413,E2 -14547.413} C_VEL
LIN {X 0,Y 333.711,Z 151.916,A -85,B 0,C 180,E1 -14551.028,E2 -14551.028} C_VEL
LIN {X 0,Y 333.736,Z 151.912,A -85,B 0,C 180,E1 -14553.753,E2 -14553.753} C_VEL
LIN {X 0,Y 333.657,Z 151.921,A -85,B 0,C 180,E1 -14557.719,E2 -14557.719} C_VEL
LIN {X 0,Y 333.74,Z 151.909,A -85,B 0,C 180,E1 -14561.586,E2 -14561.586} C_VEL
LIN {X 0,Y 333.808,Z 151.902,A -85,B 0,C 180,E1 -14565.576,E2 -14565.576} C_VEL
LIN {X 0,Y 333.818,Z 151.904,A -85,B 0,C 180,E1 -14569.077,E2 -14569.077} C_VEL
LIN {X 0,Y 333.962,Z 151.887,A -85,B 0,C 180,E1 -14572.746,E2 -14572.746} C_VEL
LIN {X 0,Y 333.803,Z 151.904,A -85,B 0,C 180,E1 -14575.169,E2 -14575.169} C_VEL
LIN {X 0,Y 334.105,Z 151.864,A -85,B 0,C 180,E1 -14577.589,E2 -14577.589} C_VEL
LIN {X 0,Y 334.245,Z 151.847,A -85,B 0,C 180,E1 -14580,E2 -14580} C_VEL
LIN {X 0,Y 334.106,Z 151.867,A -85,B 0,C 180,E1 -14582.411,E2 -14582.411} C_VEL
LIN {X 0,Y 333.991,Z 151.877,A -85,B 0,C 180,E1 -14586.598,E2 -14586.598} C_VEL
LIN {X 0,Y 333.85,Z 151.896,A -85,B 0,C 180,E1 -14589.695,E2 -14589.695} C_VEL
LIN {X 0,Y 333.796,Z 151.902,A -85,B 0,C 180,E1 -14593.391,E2 -14593.391} C_VEL
LIN {X 0,Y 333.746,Z 151.909,A -85,B 0,C 180,E1 -14597.146,E2 -14597.146} C_VEL
LIN {X 0,Y 333.732,Z 151.912,A -85,B 0,C 180,E1 -14599.69,E2 -14599.69} C_VEL
LIN {X 0,Y 333.669,Z 151.919,A -85,B 0,C 180,E1 -14603.59,E2 -14603.59} C_VEL
LIN {X 0,Y 333.734,Z 151.915,A -85,B 0,C 180,E1 -14606.246,E2 -14606.246} C_VEL
LIN {X 0,Y 333.689,Z 151.916,A -85,B 0,C 180,E1 -14608.974,E2 -14608.974} C_VEL
LIN {X 0,Y 333.645,Z 151.922,A -85,B 0,C 180,E1 -14612.588,E2 -14612.588} C_VEL
LIN {X 0,Y 333.675,Z 151.921,A -85,B 0,C 180,E1 -14616.139,E2 -14616.139} C_VEL
LIN {X 0,Y 333.646,Z 151.922,A -85,B 0,C 180,E1 -14619.192,E2 -14619.192} C_VEL
LIN {X 0,Y 333.631,Z 151.923,A -85,B 0,C 180,E1 -14622.5,E2 -14622.5} C_VEL
LIN {X 0,Y 333.595,Z 151.93,A -85,B 0,C 180,E1 -14625.955,E2 -14625.955} C_VEL
LIN {X 0,Y 333.646,Z 151.925,A -85,B 0,C 180,E1 -14629.315,E2 -14629.315} C_VEL
LIN {X 0,Y 333.664,Z 151.922,A -85,B 0,C 180,E1 -14633.168,E2 -14633.168} C_VEL
LIN {X 0,Y 333.673,Z 151.923,A -85,B 0,C 180,E1 -14635.341,E2 -14635.341} C_VEL
LIN {X 0,Y 333.702,Z 151.917,A -85,B 0,C 180,E1 -14639.71,E2 -14639.71} C_VEL
LIN {X 0,Y 333.742,Z 151.91,A -85,B 0,C 180,E1 -14642.401,E2 -14642.401} C_VEL
LIN {X 0,Y 333.725,Z 151.916,A -85,B 0,C 180,E1 -14645.091,E2 -14645.091} C_VEL
LIN {X 0,Y 333.67,Z 151.923,A -85,B 0,C 180,E1 -14649.019,E2 -14649.019} C_VEL
LIN {X 0,Y 333.74,Z 151.911,A -85,B 0,C 180,E1 -14651.587,E2 -14651.587} C_VEL
LIN {X 0,Y 333.808,Z 151.902,A -85,B 0,C 180,E1 -14655.577,E2 -14655.577} C_VEL
LIN {X 0,Y 333.817,Z 151.904,A -85,B 0,C 180,E1 -14659.078,E2 -14659.078} C_VEL
LIN {X 0,Y 333.963,Z 151.887,A -85,B 0,C 180,E1 -14662.746,E2 -14662.746} C_VEL
LIN {X 0,Y 333.803,Z 151.906,A -85,B 0,C 180,E1 -14665.169,E2 -14665.169} C_VEL
LIN {X 0,Y 333.843,Z 152.077,A -85,B 0,C 180,E1 -14666.077,E2 -14666.077} C_VEL
LIN {X 0,Y 334.844,Z 156.211,A -85,B 0,C 180,E1 -14667.241,E2 -14667.241} C_VEL
LIN {X 0,Y 340.334,Z 172.911,A -85,B 0,C 180,E1 -14667.934,E2 -14667.934} C_VEL
LIN {X 0,Y 342.039,Z 183.027,A -85,B 0,C 180,E1 -14668.256,E2 -14668.256} C_VEL
LIN {X 0,Y 340.353,Z 264.021,A -85,B 0,C 180,E1 -14670,E2 -14670} C_VEL
LIN {X 0,Y 339.829,Z 277.715,A -85,B 0,C 180,E1 -14670.556,E2 -14670.556} C_VEL
LIN {X 0,Y 339.173,Z 290.545,A -85,B 0,C 180,E1 -14671.336,E2 -14671.336} C_VEL
LIN {X 0,Y 338.357,Z 301.562,A -85,B 0,C 180,E1 -14672.232,E2 -14672.232} C_VEL
LIN {X 0,Y 337.373,Z 312.976,A -85,B 0,C 180,E1 -14673.42,E2 -14673.42} C_VEL
LIN {X 0,Y 336.297,Z 323.514,A -85,B 0,C 180,E1 -14674.795,E2 -14674.795} C_VEL
LIN {X 0,Y 335.284,Z 332.84,A -85,B 0,C 180,E1 -14676.318,E2 -14676.318} C_VEL
LIN {X 0,Y 334.329,Z 341.901,A -85,B 0,C 180,E1 -14678.158,E2 -14678.158} C_VEL
LIN {X 0,Y 333.535,Z 349.172,A -85,B 0,C 180,E1 -14680.011,E2 -14680.011} C_VEL
LIN {X 0,Y 332.871,Z 355.779,A -85,B 0,C 180,E1 -14682.189,E2 -14682.189} C_VEL
LIN {X 0,Y 332.488,Z 359.996,A -85,B 0,C 180,E1 -14684.006,E2 -14684.006} C_VEL
LIN {X 0,Y 332.102,Z 363.373,A -85,B 0,C 180,E1 -14685.969,E2 -14685.969} C_VEL
LIN {X 0,Y 331.977,Z 365.397,A -85,B 0,C 180,E1 -14687.701,E2 -14687.701} C_VEL
LIN {X 0,Y 331.898,Z 366.756,A -85,B 0,C 180,E1 -14689.804,E2 -14689.804} C_VEL
LIN {X 0,Y 331.997,Z 366.993,A -85,B 0,C 180,E1 -14691.341,E2 -14691.341} C_VEL
LIN {X 0,Y 332.196,Z 366.132,A -85,B 0,C 180,E1 -14693.701,E2 -14693.701} C_VEL
LIN {X 0,Y 332.433,Z 365.025,A -85,B 0,C 180,E1 -14695.013,E2 -14695.013} C_VEL
LIN {X 0,Y 332.922,Z 362.443,A -85,B 0,C 180,E1 -14696.972,E2 -14696.972} C_VEL
LIN {X 0,Y 333.628,Z 358.597,A -85,B 0,C 180,E1 -14698.98,E2 -14698.98} C_VEL
LIN {X 0,Y 334.518,Z 353.44,A -85,B 0,C 180,E1 -14700.981,E2 -14700.981} C_VEL
LIN {X 0,Y 335.73,Z 346.782,A -85,B 0,C 180,E1 -14702.975,E2 -14702.975} C_VEL
LIN {X 0,Y 336.933,Z 339.818,A -85,B 0,C 180,E1 -14704.639,E2 -14704.639} C_VEL
LIN {X 0,Y 338.423,Z 331.099,A -85,B 0,C 180,E1 -14706.312,E2 -14706.312} C_VEL
LIN {X 0,Y 339.891,Z 321.676,A -85,B 0,C 180,E1 -14707.775,E2 -14707.775} C_VEL
LIN {X 0,Y 341.339,Z 311.63,A -85,B 0,C 180,E1 -14709.034,E2 -14709.034} C_VEL
LIN {X 0,Y 342.861,Z 299.612,A -85,B 0,C 180,E1 -14710.218,E2 -14710.218} C_VEL
LIN {X 0,Y 343.39,Z 293.952,A -85,B 0,C 180,E1 -14710.68,E2 -14710.68} C_VEL
LIN {X 0,Y 343.359,Z 288.62,A -85,B 0,C 180,E1 -14711.106,E2 -14711.106} C_VEL
LIN {X 0,Y 341.53,Z 279.923,A -85,B 0,C 180,E1 -14711.839,E2 -14711.839} C_VEL
LIN {X 0,Y 339.476,Z 271.014,A -85,B 0,C 180,E1 -14712.473,E2 -14712.473} C_VEL
LIN {X 0,Y 339.02,Z 265.351,A -85,B 0,C 180,E1 -14712.737,E2 -14712.737} C_VEL
LIN {X 0,Y 340.743,Z 203.271,A -85,B 0,C 180,E1 -14714.124,E2 -14714.124} C_VEL
LIN {X 0,Y 341.189,Z 186.806,A -85,B 0,C 180,E1 -14714.481,E2 -14714.481} C_VEL
LIN {X 0,Y 334.168,Z 170.562,A -85,B 0,C 180,E1 -14715.564,E2 -14715.564} C_VEL
LIN {X 0,Y 327.732,Z 157.433,A -85,B 0,C 180,E1 -14716.616,E2 -14716.616} C_VEL
LIN {X 0,Y 326.549,Z 152.812,A -85,B 0,C 180,E1 -14718.254,E2 -14718.254} C_VEL
LIN {X 0,Y 326.567,Z 152.807,A -85,B 0,C 180,E1 -14721.384,E2 -14721.384} C_VEL
LIN {X 0,Y 326.618,Z 152.798,A -85,B 0,C 180,E1 -14724.852,E2 -14724.852} C_VEL
LIN {X 0,Y 326.608,Z 152.805,A -85,B 0,C 180,E1 -14727.456,E2 -14727.456} C_VEL
LIN {X 0,Y 326.581,Z 152.809,A -85,B 0,C 180,E1 -14730.333,E2 -14730.333} C_VEL
LIN {X 0,Y 326.596,Z 152.805,A -85,B 0,C 180,E1 -14733.135,E2 -14733.135} C_VEL
LIN {X 0,Y 326.59,Z 152.797,A -85,B 0,C 180,E1 -14737.211,E2 -14737.211} C_VEL
LIN {X 0,Y 326.629,Z 152.791,A -85,B 0,C 180,E1 -14741.217,E2 -14741.217} C_VEL
LIN {X 0,Y 326.715,Z 152.781,A -85,B 0,C 180,E1 -14745.467,E2 -14745.467} C_VEL
LIN {X 0,Y 326.749,Z 152.773,A -85,B 0,C 180,E1 -14748.838,E2 -14748.838} C_VEL
LIN {X 0,Y 326.914,Z 152.755,A -85,B 0,C 180,E1 -14752.589,E2 -14752.589} C_VEL
LIN {X 0,Y 326.744,Z 152.78,A -85,B 0,C 180,E1 -14755.065,E2 -14755.065} C_VEL
LIN {X 0,Y 327.002,Z 152.743,A -85,B 0,C 180,E1 -14757.537,E2 -14757.537} C_VEL
LIN {X 0,Y 327.03,Z 152.746,A -85,B 0,C 180,E1 -14761.232,E2 -14761.232} C_VEL
LIN {X 0,Y 326.75,Z 152.773,A -85,B 0,C 180,E1 -14763.7,E2 -14763.7} C_VEL
LIN {X 0,Y 326.944,Z 152.756,A -85,B 0,C 180,E1 -14766.17,E2 -14766.17} C_VEL
LIN {X 0,Y 326.785,Z 152.781,A -85,B 0,C 180,E1 -14769.907,E2 -14769.907} C_VEL
LIN {X 0,Y 326.761,Z 152.774,A -85,B 0,C 180,E1 -14773.686,E2 -14773.686} C_VEL
LIN {X 0,Y 326.666,Z 152.783,A -85,B 0,C 180,E1 -14777.53,E2 -14777.53} C_VEL
LIN {X 0,Y 326.652,Z 152.793,A -85,B 0,C 180,E1 -14780.136,E2 -14780.136} C_VEL
LIN {X 0,Y 326.636,Z 152.795,A -85,B 0,C 180,E1 -14784.13,E2 -14784.13} C_VEL
LIN {X 0,Y 326.601,Z 152.8,A -85,B 0,C 180,E1 -14788.256,E2 -14788.256} C_VEL
LIN {X 0,Y 326.576,Z 152.8,A -85,B 0,C 180,E1 -14791.097,E2 -14791.097} C_VEL
LIN {X 0,Y 326.609,Z 152.795,A -85,B 0,C 180,E1 -14794.019,E2 -14794.019} C_VEL
LIN {X 0,Y 326.625,Z 152.794,A -85,B 0,C 180,E1 -14797.238,E2 -14797.238} C_VEL
LIN {X 0,Y 326.546,Z 152.81,A -85,B 0,C 180,E1 -14801.125,E2 -14801.125} C_VEL
LIN {X 0,Y 326.563,Z 152.806,A -85,B 0,C 180,E1 -14803.526,E2 -14803.526} C_VEL
LIN {X 0,Y 326.578,Z 152.809,A -85,B 0,C 180,E1 -14807.028,E2 -14807.028} C_VEL
LIN {X 0,Y 326.613,Z 152.804,A -85,B 0,C 180,E1 -14810.773,E2 -14810.773} C_VEL
LIN {X 0,Y 326.615,Z 152.799,A -85,B 0,C 180,E1 -14814.48,E2 -14814.48} C_VEL
LIN {X 0,Y 326.665,Z 152.863,A -85,B 0,C 180,E1 -14815.17,E2 -14815.17} C_VEL
LIN {X 0,Y 329.151,Z 162.743,A -85,B 0,C 180,E1 -14818.282,E2 -14818.282} C_VEL
LIN {X 0,Y 331.388,Z 172.399,A -85,B 0,C 180,E1 -14821.152,E2 -14821.152} C_VEL
LIN {X 0,Y 332.561,Z 179.564,A -85,B 0,C 180,E1 -14823.157,E2 -14823.157} C_VEL
LIN {X 0,Y 332.174,Z 182.85,A -85,B 0,C 180,E1 -14823.957,E2 -14823.957} C_VEL
LIN {X 0,Y 337.288,Z 207.165,A -85,B 0,C 180,E1 -14825.059,E2 -14825.059} C_VEL
LIN {X 0,Y 340.153,Z 225.607,A -85,B 0,C 180,E1 -14825.774,E2 -14825.774} C_VEL
LIN {X 0,Y 338.482,Z 291.864,A -85,B 0,C 180,E1 -14827.249,E2 -14827.249} C_VEL
LIN {X 0,Y 337.47,Z 305.696,A -85,B 0,C 180,E1 -14827.783,E2 -14827.783} C_VEL
LIN {X 0,Y 336.124,Z 318.676,A -85,B 0,C 180,E1 -14828.536,E2 -14828.536} C_VEL
LIN {X 0,Y 334.545,Z 331.239,A -85,B 0,C 180,E1 -14829.558,E2 -14829.558} C_VEL
LIN {X 0,Y 332.938,Z 342.454,A -85,B 0,C 180,E1 -14830.741,E2 -14830.741} C_VEL
LIN {X 0,Y 331.254,Z 352.61,A -85,B 0,C 180,E1 -14832.083,E2 -14832.083} C_VEL
LIN {X 0,Y 329.637,Z 361.938,A -85,B 0,C 180,E1 -14833.623,E2 -14833.623} C_VEL
LIN {X 0,Y 328.258,Z 370.725,A -85,B 0,C 180,E1 -14835.43,E2 -14835.43} C_VEL
LIN {X 0,Y 326.933,Z 377.968,A -85,B 0,C 180,E1 -14837.271,E2 -14837.271} C_VEL
LIN {X 0,Y 326.13,Z 382.884,A -85,B 0,C 180,E1 -14838.817,E2 -14838.817} C_VEL
LIN {X 0,Y 325.523,Z 387.695,A -85,B 0,C 180,E1 -14840.681,E2 -14840.681} C_VEL
LIN {X 0,Y 325.11,Z 391.408,A -85,B 0,C 180,E1 -14842.547,E2 -14842.547} C_VEL
LIN {X 0,Y 324.923,Z 393.927,A -85,B 0,C 180,E1 -14844.254,E2 -14844.254} C_VEL
LIN {X 0,Y 324.935,Z 395.897,A -85,B 0,C 180,E1 -14846.279,E2 -14846.279} C_VEL
LIN {X 0,Y 324.965,Z 396.864,A -85,B 0,C 180,E1 -14848.761,E2 -14848.761} C_VEL
LIN {X 0,Y 325.044,Z 396.739,A -85,B 0,C 180,E1 -14850,E2 -14850} C_VEL
LIN {X 0,Y 324.995,Z 396.183,A -85,B 0,C 180,E1 -14851.239,E2 -14851.239} C_VEL
LIN {X 0,Y 324.955,Z 393.879,A -85,B 0,C 180,E1 -14853.72,E2 -14853.72} C_VEL
LIN {X 0,Y 324.931,Z 390.678,A -85,B 0,C 180,E1 -14855.76,E2 -14855.76} C_VEL
LIN {X 0,Y 325.081,Z 387.045,A -85,B 0,C 180,E1 -14857.453,E2 -14857.453} C_VEL
LIN {X 0,Y 325.468,Z 380.955,A -85,B 0,C 180,E1 -14859.634,E2 -14859.634} C_VEL
LIN {X 0,Y 326.041,Z 374.254,A -85,B 0,C 180,E1 -14861.501,E2 -14861.501} C_VEL
LIN {X 0,Y 326.951,Z 365.928,A -85,B 0,C 180,E1 -14863.36,E2 -14863.36} C_VEL
LIN {X 0,Y 327.851,Z 357.382,A -85,B 0,C 180,E1 -14864.906,E2 -14864.906} C_VEL
LIN {X 0,Y 328.95,Z 346.799,A -85,B 0,C 180,E1 -14866.444,E2 -14866.444} C_VEL
LIN {X 0,Y 330.135,Z 334.875,A -85,B 0,C 180,E1 -14867.819,E2 -14867.819} C_VEL
LIN {X 0,Y 331.308,Z 322.873,A -85,B 0,C 180,E1 -14868.874,E2 -14868.874} C_VEL
LIN {X 0,Y 332.325,Z 310.387,A -85,B 0,C 180,E1 -14869.697,E2 -14869.697} C_VEL
LIN {X 0,Y 333.092,Z 297.472,A -85,B 0,C 180,E1 -14870.293,E2 -14870.293} C_VEL
LIN {X 0,Y 333.556,Z 282.004,A -85,B 0,C 180,E1 -14870.706,E2 -14870.706} C_VEL
LIN {X 0,Y 334.529,Z 223.499,A -85,B 0,C 180,E1 -14871.978,E2 -14871.978} C_VEL
LIN {X 0,Y 329.205,Z 183.878,A -85,B 0,C 180,E1 -14873.207,E2 -14873.207} C_VEL
LIN {X 0,Y 330.384,Z 172.762,A -85,B 0,C 180,E1 -14875.854,E2 -14875.854} C_VEL
LIN {X 0,Y 329.602,Z 167.134,A -85,B 0,C 180,E1 -14877.285,E2 -14877.285} C_VEL
LIN {X 0,Y 327.301,Z 155.951,A -85,B 0,C 180,E1 -14880.238,E2 -14880.238} C_VEL
LIN {X 0,Y 326.643,Z 152.799,A -85,B 0,C 180,E1 -14881.134,E2 -14881.134} C_VEL
LIN {X 0,Y 326.621,Z 152.797,A -85,B 0,C 180,E1 -14885.148,E2 -14885.148} C_VEL
LIN {X 0,Y 326.624,Z 152.797,A -85,B 0,C 180,E1 -14888.608,E2 -14888.608} C_VEL
LIN {X 0,Y 326.577,Z 152.807,A -85,B 0,C 180,E1 -14891.845,E2 -14891.845} C_VEL
LIN {X 0,Y 326.528,Z 152.81,A -85,B 0,C 180,E1 -14895.257,E2 -14895.257} C_VEL
LIN {X 0,Y 326.578,Z 152.803,A -85,B 0,C 180,E1 -14898.868,E2 -14898.868} C_VEL
LIN {X 0,Y 326.628,Z 152.796,A -85,B 0,C 180,E1 -14902.761,E2 -14902.761} C_VEL
LIN {X 0,Y 326.607,Z 152.8,A -85,B 0,C 180,E1 -14905.98,E2 -14905.98} C_VEL
LIN {X 0,Y 326.661,Z 152.792,A -85,B 0,C 180,E1 -14910.341,E2 -14910.341} C_VEL
LIN {X 0,Y 326.69,Z 152.788,A -85,B 0,C 180,E1 -14914.516,E2 -14914.516} C_VEL
LIN {X 0,Y 326.618,Z 152.797,A -85,B 0,C 180,E1 -14918.543,E2 -14918.543} C_VEL
LIN {X 0,Y 326.707,Z 152.787,A -85,B 0,C 180,E1 -14921.175,E2 -14921.175} C_VEL
LIN {X 0,Y 326.763,Z 152.78,A -85,B 0,C 180,E1 -14925.433,E2 -14925.433} C_VEL
LIN {X 0,Y 326.758,Z 152.784,A -85,B 0,C 180,E1 -14928.838,E2 -14928.838} C_VEL
LIN {X 0,Y 326.918,Z 152.762,A -85,B 0,C 180,E1 -14932.589,E2 -14932.589} C_VEL
LIN {X 0,Y 326.77,Z 152.781,A -85,B 0,C 180,E1 -14935.064,E2 -14935.064} C_VEL
LIN {X 0,Y 327.045,Z 152.744,A -85,B 0,C 180,E1 -14937.536,E2 -14937.536} C_VEL
LIN {X 0,Y 327.197,Z 152.725,A -85,B 0,C 180,E1 -14940,E2 -14940} C_VEL
LIN {X 0,Y 327.046,Z 152.746,A -85,B 0,C 180,E1 -14942.463,E2 -14942.463} C_VEL
LIN {X 0,Y 326.961,Z 152.753,A -85,B 0,C 180,E1 -14946.588,E2 -14946.588} C_VEL
LIN {X 0,Y 326.805,Z 152.774,A -85,B 0,C 180,E1 -14949.906,E2 -14949.906} C_VEL
LIN {X 0,Y 326.758,Z 152.779,A -85,B 0,C 180,E1 -14953.685,E2 -14953.685} C_VEL
LIN {X 0,Y 326.698,Z 152.787,A -85,B 0,C 180,E1 -14957.528,E2 -14957.528} C_VEL
LIN {X 0,Y 326.658,Z 152.796,A -85,B 0,C 180,E1 -14960.135,E2 -14960.135} C_VEL
LIN {X 0,Y 326.648,Z 152.799,A -85,B 0,C 180,E1 -14964.129,E2 -14964.129} C_VEL
LIN {X 0,Y 326.682,Z 152.789,A -85,B 0,C 180,E1 -14966.858,E2 -14966.858} C_VEL
LIN {X 0,Y 326.633,Z 152.795,A -85,B 0,C 180,E1 -14970.61,E2 -14970.61} C_VEL
LIN {X 0,Y 326.606,Z 152.803,A -85,B 0,C 180,E1 -14974.019,E2 -14974.019} C_VEL
LIN {X 0,Y 326.626,Z 152.796,A -85,B 0,C 180,E1 -14977.239,E2 -14977.239} C_VEL
LIN {X 0,Y 326.576,Z 152.803,A -85,B 0,C 180,E1 -14981.131,E2 -14981.131} C_VEL
LIN {X 0,Y 326.526,Z 152.808,A -85,B 0,C 180,E1 -14984.743,E2 -14984.743} C_VEL
LIN {X 0,Y 326.575,Z 152.803,A -85,B 0,C 180,E1 -14988.154,E2 -14988.154} C_VEL
LIN {X 0,Y 326.622,Z 152.801,A -85,B 0,C 180,E1 -14991.391,E2 -14991.391} C_VEL
LIN {X 0,Y 326.618,Z 152.798,A -85,B 0,C 180,E1 -14994.851,E2 -14994.851} C_VEL
LIN {X 0,Y 326.606,Z 152.802,A -85,B 0,C 180,E1 -14997.456,E2 -14997.456} C_VEL
LIN {X 0,Y 326.66,Z 152.791,A -85,B 0,C 180,E1 -15000.341,E2 -15000.341} C_VEL
LIN {X 0,Y 326.689,Z 152.788,A -85,B 0,C 180,E1 -15004.516,E2 -15004.516} C_VEL
LIN {X 0,Y 326.617,Z 152.798,A -85,B 0,C 180,E1 -15008.544,E2 -15008.544} C_VEL
LIN {X 0,Y 326.706,Z 152.79,A -85,B 0,C 180,E1 -15011.175,E2 -15011.175} C_VEL
LIN {X 0,Y 326.762,Z 152.781,A -85,B 0,C 180,E1 -15015.433,E2 -15015.433} C_VEL
LIN {X 0,Y 326.758,Z 152.785,A -85,B 0,C 180,E1 -15018.839,E2 -15018.839} C_VEL
LIN {X 0,Y 326.918,Z 152.762,A -85,B 0,C 180,E1 -15022.589,E2 -15022.589} C_VEL
LIN {X 0,Y 326.77,Z 152.783,A -85,B 0,C 180,E1 -15025.065,E2 -15025.065} C_VEL
LIN {X 0,Y 326.777,Z 152.812,A -85,B 0,C 180,E1 -15025.76,E2 -15025.76} C_VEL
LIN {X 0,Y 327.65,Z 156.538,A -85,B 0,C 180,E1 -15026.822,E2 -15026.822} C_VEL
LIN {X 0,Y 333.769,Z 174.782,A -85,B 0,C 180,E1 -15027.603,E2 -15027.603} C_VEL
LIN {X 0,Y 335.266,Z 183.221,A -85,B 0,C 180,E1 -15027.88,E2 -15027.88} C_VEL
LIN {X 0,Y 333.566,Z 264.303,A -85,B 0,C 180,E1 -15029.661,E2 -15029.661} C_VEL
LIN {X 0,Y 333.026,Z 277.281,A -85,B 0,C 180,E1 -15030.189,E2 -15030.189} C_VEL
LIN {X 0,Y 332.368,Z 290.347,A -85,B 0,C 180,E1 -15030.985,E2 -15030.985} C_VEL
LIN {X 0,Y 331.445,Z 302.277,A -85,B 0,C 180,E1 -15031.975,E2 -15031.975} C_VEL
LIN {X 0,Y 330.381,Z 314.244,A -85,B 0,C 180,E1 -15033.26,E2 -15033.26} C_VEL
LIN {X 0,Y 329.348,Z 324.075,A -85,B 0,C 180,E1 -15034.59,E2 -15034.59} C_VEL
LIN {X 0,Y 328.272,Z 333.368,A -85,B 0,C 180,E1 -15036.145,E2 -15036.145} C_VEL
LIN {X 0,Y 327.301,Z 342.298,A -85,B 0,C 180,E1 -15038.002,E2 -15038.002} C_VEL
LIN {X 0,Y 326.489,Z 349.619,A -85,B 0,C 180,E1 -15039.916,E2 -15039.916} C_VEL
LIN {X 0,Y 325.867,Z 355.373,A -85,B 0,C 180,E1 -15041.823,E2 -15041.823} C_VEL
LIN {X 0,Y 325.458,Z 359.881,A -85,B 0,C 180,E1 -15043.741,E2 -15043.741} C_VEL
LIN {X 0,Y 325.202,Z 362.276,A -85,B 0,C 180,E1 -15045.031,E2 -15045.031} C_VEL
LIN {X 0,Y 324.984,Z 364.199,A -85,B 0,C 180,E1 -15046.328,E2 -15046.328} C_VEL
LIN {X 0,Y 324.873,Z 365.832,A -85,B 0,C 180,E1 -15047.852,E2 -15047.852} C_VEL
LIN {X 0,Y 324.837,Z 367.213,A -85,B 0,C 180,E1 -15050.253,E2 -15050.253} C_VEL
LIN {X 0,Y 324.924,Z 367.308,A -85,B 0,C 180,E1 -15051.574,E2 -15051.574} C_VEL
LIN {X 0,Y 324.994,Z 366.983,A -85,B 0,C 180,E1 -15052.908,E2 -15052.908} C_VEL
LIN {X 0,Y 325.339,Z 365.66,A -85,B 0,C 180,E1 -15054.867,E2 -15054.867} C_VEL
LIN {X 0,Y 325.83,Z 363.182,A -85,B 0,C 180,E1 -15056.934,E2 -15056.934} C_VEL
LIN {X 0,Y 326.554,Z 359.582,A -85,B 0,C 180,E1 -15058.963,E2 -15058.963} C_VEL
LIN {X 0,Y 327.477,Z 354.65,A -85,B 0,C 180,E1 -15061.002,E2 -15061.002} C_VEL
LIN {X 0,Y 328.667,Z 348.402,A -85,B 0,C 180,E1 -15062.985,E2 -15062.985} C_VEL
LIN {X 0,Y 329.946,Z 341.489,A -85,B 0,C 180,E1 -15064.736,E2 -15064.736} C_VEL
LIN {X 0,Y 331.473,Z 333.259,A -85,B 0,C 180,E1 -15066.418,E2 -15066.418} C_VEL
LIN {X 0,Y 332.964,Z 324.182,A -85,B 0,C 180,E1 -15067.925,E2 -15067.925} C_VEL
LIN {X 0,Y 334.549,Z 314.123,A -85,B 0,C 180,E1 -15069.261,E2 -15069.261} C_VEL
LIN {X 0,Y 336.029,Z 303.231,A -85,B 0,C 180,E1 -15070.418,E2 -15070.418} C_VEL
LIN {X 0,Y 337.319,Z 290.708,A -85,B 0,C 180,E1 -15071.459,E2 -15071.459} C_VEL
LIN {X 0,Y 338.351,Z 277.749,A -85,B 0,C 180,E1 -15072.233,E2 -15072.233} C_VEL
LIN {X 0,Y 339.02,Z 265.351,A -85,B 0,C 180,E1 -15072.737,E2 -15072.737} C_VEL
LIN {X 0,Y 338.584,Z 259.61,A -85,B 0,C 180,E1 -15072.969,E2 -15072.969} C_VEL
LIN {X 0,Y 334.09,Z 240.97,A -85,B 0,C 180,E1 -15073.827,E2 -15073.827} C_VEL
LIN {X 0,Y 333.654,Z 235.171,A -85,B 0,C 180,E1 -15074.003,E2 -15074.003} C_VEL
LIN {X 0,Y 334.977,Z 188.812,A -85,B 0,C 180,E1 -15075.027,E2 -15075.027} C_VEL
LIN {X 0,Y 328.722,Z 174.219,A -85,B 0,C 180,E1 -15076.039,E2 -15076.039} C_VEL
LIN {X 0,Y 321.885,Z 160.635,A -85,B 0,C 180,E1 -15077.145,E2 -15077.145} C_VEL
LIN {X 0,Y 320.583,Z 157.909,A -85,B 0,C 180,E1 -15077.376,E2 -15077.376} C_VEL
LIN {X 0,Y 319.512,Z 153.691,A -85,B 0,C 180,E1 -15078.919,E2 -15078.919} C_VEL
LIN {X 0,Y 319.541,Z 153.679,A -85,B 0,C 180,E1 -15082.353,E2 -15082.353} C_VEL
LIN {X 0,Y 319.559,Z 153.68,A -85,B 0,C 180,E1 -15085.124,E2 -15085.124} C_VEL
LIN {X 0,Y 319.524,Z 153.686,A -85,B 0,C 180,E1 -15088.138,E2 -15088.138} C_VEL
LIN {X 0,Y 319.545,Z 153.68,A -85,B 0,C 180,E1 -15091.613,E2 -15091.613} C_VEL
LIN {X 0,Y 319.526,Z 153.686,A -85,B 0,C 180,E1 -15095.298,E2 -15095.298} C_VEL
LIN {X 0,Y 319.56,Z 153.673,A -85,B 0,C 180,E1 -15098.045,E2 -15098.045} C_VEL
LIN {X 0,Y 319.574,Z 153.673,A -85,B 0,C 180,E1 -15102.068,E2 -15102.068} C_VEL
LIN {X 0,Y 319.694,Z 153.658,A -85,B 0,C 180,E1 -15106.006,E2 -15106.006} C_VEL
LIN {X 0,Y 319.732,Z 153.649,A -85,B 0,C 180,E1 -15109.872,E2 -15109.872} C_VEL
LIN {X 0,Y 319.899,Z 153.626,A -85,B 0,C 180,E1 -15113.694,E2 -15113.694} C_VEL
LIN {X 0,Y 319.948,Z 153.622,A -85,B 0,C 180,E1 -15117.482,E2 -15117.482} C_VEL
LIN {X 0,Y 319.999,Z 153.622,A -85,B 0,C 180,E1 -15121.259,E2 -15121.259} C_VEL
LIN {X 0,Y 319.7,Z 153.651,A -85,B 0,C 180,E1 -15123.782,E2 -15123.782} C_VEL
LIN {X 0,Y 319.901,Z 153.632,A -85,B 0,C 180,E1 -15126.307,E2 -15126.307} C_VEL
LIN {X 0,Y 319.737,Z 153.657,A -85,B 0,C 180,E1 -15130.128,E2 -15130.128} C_VEL
LIN {X 0,Y 319.734,Z 153.652,A -85,B 0,C 180,E1 -15133.992,E2 -15133.992} C_VEL
LIN {X 0,Y 319.626,Z 153.659,A -85,B 0,C 180,E1 -15137.929,E2 -15137.929} C_VEL
LIN {X 0,Y 319.6,Z 153.673,A -85,B 0,C 180,E1 -15140.6,E2 -15140.6} C_VEL
LIN {X 0,Y 319.556,Z 153.673,A -85,B 0,C 180,E1 -15143.321,E2 -15143.321} C_VEL
LIN {X 0,Y 319.572,Z 153.669,A -85,B 0,C 180,E1 -15146.094,E2 -15146.094} C_VEL
LIN {X 0,Y 319.545,Z 153.681,A -85,B 0,C 180,E1 -15148.938,E2 -15148.938} C_VEL
LIN {X 0,Y 319.526,Z 153.682,A -85,B 0,C 180,E1 -15151.863,E2 -15151.863} C_VEL
LIN {X 0,Y 319.582,Z 153.676,A -85,B 0,C 180,E1 -15155.543,E2 -15155.543} C_VEL
LIN {X 0,Y 319.53,Z 153.683,A -85,B 0,C 180,E1 -15159.662,E2 -15159.662} C_VEL
LIN {X 0,Y 319.522,Z 153.683,A -85,B 0,C 180,E1 -15163.46,E2 -15163.46} C_VEL
LIN {X 0,Y 319.556,Z 153.684,A -85,B 0,C 180,E1 -15167.017,E2 -15167.017} C_VEL
LIN {X 0,Y 319.549,Z 153.682,A -85,B 0,C 180,E1 -15170.371,E2 -15170.371} C_VEL
LIN {X 0,Y 319.594,Z 153.675,A -85,B 0,C 180,E1 -15174.454,E2 -15174.454} C_VEL
LIN {X 0,Y 322.123,Z 163.54,A -85,B 0,C 180,E1 -15177.687,E2 -15177.687} C_VEL
LIN {X 0,Y 324.517,Z 173.895,A -85,B 0,C 180,E1 -15180.849,E2 -15180.849} C_VEL
LIN {X 0,Y 325.592,Z 179.767,A -85,B 0,C 180,E1 -15182.547,E2 -15182.547} C_VEL
LIN {X 0,Y 325.614,Z 182.328,A -85,B 0,C 180,E1 -15183.233,E2 -15183.233} C_VEL
LIN {X 0,Y 329.725,Z 201.427,A -85,B 0,C 180,E1 -15184.177,E2 -15184.177} C_VEL
LIN {X 0,Y 332.814,Z 218.801,A -85,B 0,C 180,E1 -15184.92,E2 -15184.92} C_VEL
LIN {X 0,Y 333.934,Z 226.945,A -85,B 0,C 180,E1 -15185.23,E2 -15185.23} C_VEL
LIN {X 0,Y 332.152,Z 292.077,A -85,B 0,C 180,E1 -15186.708,E2 -15186.708} C_VEL
LIN {X 0,Y 331.102,Z 305.729,A -85,B 0,C 180,E1 -15187.25,E2 -15187.25} C_VEL
LIN {X 0,Y 329.684,Z 318.594,A -85,B 0,C 180,E1 -15188.013,E2 -15188.013} C_VEL
LIN {X 0,Y 328.13,Z 330.317,A -85,B 0,C 180,E1 -15188.976,E2 -15188.976} C_VEL
LIN {X 0,Y 326.461,Z 341.637,A -85,B 0,C 180,E1 -15190.18,E2 -15190.18} C_VEL
LIN {X 0,Y 324.693,Z 351.892,A -85,B 0,C 180,E1 -15191.545,E2 -15191.545} C_VEL
LIN {X 0,Y 322.936,Z 361.502,A -85,B 0,C 180,E1 -15193.151,E2 -15193.151} C_VEL
LIN {X 0,Y 321.567,Z 369.459,A -85,B 0,C 180,E1 -15194.795,E2 -15194.795} C_VEL
LIN {X 0,Y 320.248,Z 376.864,A -85,B 0,C 180,E1 -15196.678,E2 -15196.678} C_VEL
LIN {X 0,Y 319.125,Z 382.837,A -85,B 0,C 180,E1 -15198.568,E2 -15198.568} C_VEL
LIN {X 0,Y 318.474,Z 387.582,A -85,B 0,C 180,E1 -15200.473,E2 -15200.473} C_VEL
LIN {X 0,Y 318.033,Z 391.235,A -85,B 0,C 180,E1 -15202.38,E2 -15202.38} C_VEL
LIN {X 0,Y 317.833,Z 393.908,A -85,B 0,C 180,E1 -15204.3,E2 -15204.3} C_VEL
LIN {X 0,Y 317.838,Z 395.625,A -85,B 0,C 180,E1 -15206.196,E2 -15206.196} C_VEL
LIN {X 0,Y 317.868,Z 396.547,A -85,B 0,C 180,E1 -15208.733,E2 -15208.733} C_VEL
LIN {X 0,Y 317.953,Z 396.381,A -85,B 0,C 180,E1 -15210,E2 -15210} C_VEL
LIN {X 0,Y 317.9,Z 395.803,A -85,B 0,C 180,E1 -15211.267,E2 -15211.267} C_VEL
LIN {X 0,Y 317.844,Z 394.83,A -85,B 0,C 180,E1 -15212.534,E2 -15212.534} C_VEL
LIN {X 0,Y 317.88,Z 393.454,A -85,B 0,C 180,E1 -15213.803,E2 -15213.803} C_VEL
LIN {X 0,Y 317.856,Z 390.465,A -85,B 0,C 180,E1 -15215.741,E2 -15215.741} C_VEL
LIN {X 0,Y 318.009,Z 386.523,A -85,B 0,C 180,E1 -15217.62,E2 -15217.62} C_VEL
LIN {X 0,Y 318.431,Z 380.352,A -85,B 0,C 180,E1 -15219.849,E2 -15219.849} C_VEL
LIN {X 0,Y 319.024,Z 373.587,A -85,B 0,C 180,E1 -15221.758,E2 -15221.758} C_VEL
LIN {X 0,Y 319.952,Z 365.184,A -85,B 0,C 180,E1 -15223.658,E2 -15223.658} C_VEL
LIN {X 0,Y 320.886,Z 356.507,A -85,B 0,C 180,E1 -15225.237,E2 -15225.237} C_VEL
LIN {X 0,Y 322.068,Z 345.794,A -85,B 0,C 180,E1 -15226.806,E2 -15226.806} C_VEL
LIN {X 0,Y 323.178,Z 335.159,A -85,B 0,C 180,E1 -15228.052,E2 -15228.052} C_VEL
LIN {X 0,Y 324.388,Z 323.379,A -85,B 0,C 180,E1 -15229.128,E2 -15229.128} C_VEL
LIN {X 0,Y 325.407,Z 311.128,A -85,B 0,C 180,E1 -15229.969,E2 -15229.969} C_VEL
LIN {X 0,Y 326.27,Z 297.78,A -85,B 0,C 180,E1 -15230.613,E2 -15230.613} C_VEL
LIN {X 0,Y 326.723,Z 282.756,A -85,B 0,C 180,E1 -15231.036,E2 -15231.036} C_VEL
LIN {X 0,Y 327.691,Z 223.749,A -85,B 0,C 180,E1 -15232.346,E2 -15232.346} C_VEL
LIN {X 0,Y 322.35,Z 183.616,A -85,B 0,C 180,E1 -15233.617,E2 -15233.617} C_VEL
LIN {X 0,Y 323.412,Z 173.497,A -85,B 0,C 180,E1 -15236.073,E2 -15236.073} C_VEL
LIN {X 0,Y 321.931,Z 164.839,A -85,B 0,C 180,E1 -15238.347,E2 -15238.347} C_VEL
LIN {X 0,Y 319.594,Z 153.676,A -85,B 0,C 180,E1 -15241.421,E2 -15241.421} C_VEL
LIN {X 0,Y 319.581,Z 153.677,A -85,B 0,C 180,E1 -15245.543,E2 -15245.543} C_VEL
LIN {X 0,Y 319.574,Z 153.679,A -85,B 0,C 180,E1 -15248.008,E2 -15248.008} C_VEL
LIN {X 0,Y 319.527,Z 153.684,A -85,B 0,C 180,E1 -15251.597,E2 -15251.597} C_VEL
LIN {X 0,Y 319.489,Z 153.687,A -85,B 0,C 180,E1 -15255.257,E2 -15255.257} C_VEL
LIN {X 0,Y 319.529,Z 153.681,A -85,B 0,C 180,E1 -15258.711,E2 -15258.711} C_VEL
LIN {X 0,Y 319.562,Z 153.677,A -85,B 0,C 180,E1 -15262.348,E2 -15262.348} C_VEL
LIN {X 0,Y 319.56,Z 153.679,A -85,B 0,C 180,E1 -15265.123,E2 -15265.123} C_VEL
LIN {X 0,Y 319.57,Z 153.678,A -85,B 0,C 180,E1 -15269.058,E2 -15269.058} C_VEL
LIN {X 0,Y 319.609,Z 153.67,A -85,B 0,C 180,E1 -15272.498,E2 -15272.498} C_VEL
LIN {X 0,Y 319.604,Z 153.676,A -85,B 0,C 180,E1 -15275.304,E2 -15275.304} C_VEL
LIN {X 0,Y 319.586,Z 153.673,A -85,B 0,C 180,E1 -15279.399,E2 -15279.399} C_VEL
LIN {X 0,Y 319.624,Z 153.662,A -85,B 0,C 180,E1 -15282.071,E2 -15282.071} C_VEL
LIN {X 0,Y 319.732,Z 153.653,A -85,B 0,C 180,E1 -15286.008,E2 -15286.008} C_VEL
LIN {X 0,Y 319.735,Z 153.654,A -85,B 0,C 180,E1 -15289.872,E2 -15289.872} C_VEL
LIN {X 0,Y 319.907,Z 153.631,A -85,B 0,C 180,E1 -15293.693,E2 -15293.693} C_VEL
LIN {X 0,Y 319.989,Z 153.623,A -85,B 0,C 180,E1 -15297.482,E2 -15297.482} C_VEL
LIN {X 0,Y 320.149,Z 153.603,A -85,B 0,C 180,E1 -15300,E2 -15300} C_VEL
LIN {X 0,Y 319.99,Z 153.625,A -85,B 0,C 180,E1 -15302.517,E2 -15302.517} C_VEL
LIN {X 0,Y 319.923,Z 153.631,A -85,B 0,C 180,E1 -15306.575,E2 -15306.575} C_VEL
LIN {X 0,Y 319.752,Z 153.654,A -85,B 0,C 180,E1 -15310.127,E2 -15310.127} C_VEL
LIN {X 0,Y 319.73,Z 153.657,A -85,B 0,C 180,E1 -15314.724,E2 -15314.724} C_VEL
LIN {X 0,Y 319.688,Z 153.66,A -85,B 0,C 180,E1 -15319.037,E2 -15319.037} C_VEL
LIN {X 0,Y 319.559,Z 153.676,A -85,B 0,C 180,E1 -15323.32,E2 -15323.32} C_VEL
LIN {X 0,Y 319.633,Z 153.673,A -85,B 0,C 180,E1 -15326.088,E2 -15326.088} C_VEL
LIN {X 0,Y 319.578,Z 153.673,A -85,B 0,C 180,E1 -15328.934,E2 -15328.934} C_VEL
LIN {X 0,Y 319.53,Z 153.683,A -85,B 0,C 180,E1 -15331.862,E2 -15331.862} C_VEL
LIN {X 0,Y 319.579,Z 153.676,A -85,B 0,C 180,E1 -15335.543,E2 -15335.543} C_VEL
LIN {X 0,Y 319.557,Z 153.679,A -85,B 0,C 180,E1 -15339.669,E2 -15339.669} C_VEL
LIN {X 0,Y 319.52,Z 153.684,A -85,B 0,C 180,E1 -15343.461,E2 -15343.461} C_VEL
LIN {X 0,Y 319.553,Z 153.677,A -85,B 0,C 180,E1 -15347.017,E2 -15347.017} C_VEL
LIN {X 0,Y 319.545,Z 153.678,A -85,B 0,C 180,E1 -15350.371,E2 -15350.371} C_VEL
LIN {X 0,Y 319.557,Z 153.681,A -85,B 0,C 180,E1 -15353.572,E2 -15353.572} C_VEL
LIN {X 0,Y 319.576,Z 153.674,A -85,B 0,C 180,E1 -15356.687,E2 -15356.687} C_VEL
LIN {X 0,Y 319.59,Z 153.675,A -85,B 0,C 180,E1 -15359.617,E2 -15359.617} C_VEL
LIN {X 0,Y 319.607,Z 153.671,A -85,B 0,C 180,E1 -15362.498,E2 -15362.498} C_VEL
LIN {X 0,Y 319.603,Z 153.674,A -85,B 0,C 180,E1 -15365.304,E2 -15365.304} C_VEL
LIN {X 0,Y 319.586,Z 153.676,A -85,B 0,C 180,E1 -15369.399,E2 -15369.399} C_VEL
LIN {X 0,Y 319.624,Z 153.668,A -85,B 0,C 180,E1 -15372.071,E2 -15372.071} C_VEL
LIN {X 0,Y 319.732,Z 153.655,A -85,B 0,C 180,E1 -15376.008,E2 -15376.008} C_VEL
LIN {X 0,Y 319.735,Z 153.655,A -85,B 0,C 180,E1 -15379.872,E2 -15379.872} C_VEL
LIN {X 0,Y 319.907,Z 153.634,A -85,B 0,C 180,E1 -15383.694,E2 -15383.694} C_VEL
LIN {X 0,Y 319.752,Z 153.81,A -85,B 0,C 180,E1 -15385.509,E2 -15385.509} C_VEL
LIN {X 0,Y 320.364,Z 156.66,A -85,B 0,C 180,E1 -15386.368,E2 -15386.368} C_VEL
LIN {X 0,Y 326.597,Z 174.562,A -85,B 0,C 180,E1 -15387.18,E2 -15387.18} C_VEL
LIN {X 0,Y 328.295,Z 182.638,A -85,B 0,C 180,E1 -15387.47,E2 -15387.47} C_VEL
LIN {X 0,Y 328.405,Z 191.336,A -85,B 0,C 180,E1 -15387.677,E2 -15387.677} C_VEL
LIN {X 0,Y 326.774,Z 264.219,A -85,B 0,C 180,E1 -15389.307,E2 -15389.307} C_VEL
LIN {X 0,Y 326.208,Z 278.065,A -85,B 0,C 180,E1 -15389.885,E2 -15389.885} C_VEL
LIN {X 0,Y 325.498,Z 291.002,A -85,B 0,C 180,E1 -15390.696,E2 -15390.696} C_VEL
LIN {X 0,Y 324.534,Z 302.875,A -85,B 0,C 180,E1 -15391.707,E2 -15391.707} C_VEL
LIN {X 0,Y 323.559,Z 313.706,A -85,B 0,C 180,E1 -15392.888,E2 -15392.888} C_VEL
LIN {X 0,Y 322.37,Z 324.582,A -85,B 0,C 180,E1 -15394.376,E2 -15394.376} C_VEL
LIN {X 0,Y 321.26,Z 333.851,A -85,B 0,C 180,E1 -15395.965,E2 -15395.965} C_VEL
LIN {X 0,Y 320.272,Z 342.621,A -85,B 0,C 180,E1 -15397.829,E2 -15397.829} C_VEL
LIN {X 0,Y 319.445,Z 350.045,A -85,B 0,C 180,E1 -15399.817,E2 -15399.817} C_VEL
LIN {X 0,Y 318.734,Z 356.614,A -85,B 0,C 180,E1 -15402.092,E2 -15402.092} C_VEL
LIN {X 0,Y 318.315,Z 360.922,A -85,B 0,C 180,E1 -15404.056,E2 -15404.056} C_VEL
LIN {X 0,Y 318.059,Z 363.183,A -85,B 0,C 180,E1 -15405.377,E2 -15405.377} C_VEL
LIN {X 0,Y 317.855,Z 364.95,A -85,B 0,C 180,E1 -15406.705,E2 -15406.705} C_VEL
LIN {X 0,Y 317.777,Z 366.285,A -85,B 0,C 180,E1 -15408.037,E2 -15408.037} C_VEL
LIN {X 0,Y 317.726,Z 367.174,A -85,B 0,C 180,E1 -15409.378,E2 -15409.378} C_VEL
LIN {X 0,Y 317.848,Z 367.629,A -85,B 0,C 180,E1 -15411.772,E2 -15411.772} C_VEL
LIN {X 0,Y 317.99,Z 367.155,A -85,B 0,C 180,E1 -15413.442,E2 -15413.442} C_VEL
LIN {X 0,Y 318.324,Z 365.925,A -85,B 0,C 180,E1 -15415.15,E2 -15415.15} C_VEL
LIN {X 0,Y 318.944,Z 362.945,A -85,B 0,C 180,E1 -15417.564,E2 -15417.564} C_VEL
LIN {X 0,Y 319.75,Z 359.095,A -85,B 0,C 180,E1 -15419.64,E2 -15419.64} C_VEL
LIN {X 0,Y 320.82,Z 353.912,A -85,B 0,C 180,E1 -15421.719,E2 -15421.719} C_VEL
LIN {X 0,Y 322.01,Z 347.971,A -85,B 0,C 180,E1 -15423.583,E2 -15423.583} C_VEL
LIN {X 0,Y 323.551,Z 340.192,A -85,B 0,C 180,E1 -15425.525,E2 -15425.525} C_VEL
LIN {X 0,Y 325.161,Z 331.514,A -85,B 0,C 180,E1 -15427.243,E2 -15427.243} C_VEL
LIN {X 0,Y 326.932,Z 321.361,A -85,B 0,C 180,E1 -15428.855,E2 -15428.855} C_VEL
LIN {X 0,Y 328.532,Z 311.362,A -85,B 0,C 180,E1 -15430.124,E2 -15430.124} C_VEL
LIN {X 0,Y 330.086,Z 299.566,A -85,B 0,C 180,E1 -15431.303,E2 -15431.303} C_VEL
LIN {X 0,Y 331.308,Z 287.431,A -85,B 0,C 180,E1 -15432.236,E2 -15432.236} C_VEL
LIN {X 0,Y 332.229,Z 275.379,A -85,B 0,C 180,E1 -15432.914,E2 -15432.914} C_VEL
LIN {X 0,Y 332.853,Z 262.617,A -85,B 0,C 180,E1 -15433.384,E2 -15433.384} C_VEL
LIN {X 0,Y 333.654,Z 235.171,A -85,B 0,C 180,E1 -15434.003,E2 -15434.003} C_VEL
LIN {X 0,Y 333.217,Z 229.375,A -85,B 0,C 180,E1 -15434.189,E2 -15434.189} C_VEL
LIN {X 0,Y 328.768,Z 210.761,A -85,B 0,C 180,E1 -15435.097,E2 -15435.097} C_VEL
LIN {X 0,Y 328.342,Z 204.966,A -85,B 0,C 180,E1 -15435.288,E2 -15435.288} C_VEL
LIN {X 0,Y 328.752,Z 190.495,A -85,B 0,C 180,E1 -15435.617,E2 -15435.617} C_VEL
LIN {X 0,Y 322.142,Z 175.412,A -85,B 0,C 180,E1 -15436.723,E2 -15436.723} C_VEL
LIN {X 0,Y 315.141,Z 161.696,A -85,B 0,C 180,E1 -15437.9,E2 -15437.9} C_VEL
LIN {X 0,Y 313.417,Z 158.256,A -85,B 0,C 180,E1 -15438.224,E2 -15438.224} C_VEL
LIN {X 0,Y 312.489,Z 154.557,A -85,B 0,C 180,E1 -15439.641,E2 -15439.641} C_VEL
LIN {X 0,Y 312.533,Z 154.544,A -85,B 0,C 180,E1 -15444.051,E2 -15444.051} C_VEL
LIN {X 0,Y 312.501,Z 154.562,A -85,B 0,C 180,E1 -15447.334,E2 -15447.334} C_VEL
LIN {X 0,Y 312.485,Z 154.559,A -85,B 0,C 180,E1 -15451.299,E2 -15451.299} C_VEL
LIN {X 0,Y 312.517,Z 154.555,A -85,B 0,C 180,E1 -15454.705,E2 -15454.705} C_VEL
LIN {X 0,Y 312.538,Z 154.547,A -85,B 0,C 180,E1 -15457.526,E2 -15457.526} C_VEL
LIN {X 0,Y 312.54,Z 154.547,A -85,B 0,C 180,E1 -15461.651,E2 -15461.651} C_VEL
LIN {X 0,Y 312.638,Z 154.535,A -85,B 0,C 180,E1 -15465.684,E2 -15465.684} C_VEL
LIN {X 0,Y 312.682,Z 154.525,A -85,B 0,C 180,E1 -15469.641,E2 -15469.641} C_VEL
LIN {X 0,Y 312.797,Z 154.516,A -85,B 0,C 180,E1 -15472.253,E2 -15472.253} C_VEL
LIN {X 0,Y 312.685,Z 154.532,A -85,B 0,C 180,E1 -15474.842,E2 -15474.842} C_VEL
LIN {X 0,Y 312.967,Z 154.49,A -85,B 0,C 180,E1 -15478.714,E2 -15478.714} C_VEL
LIN {X 0,Y 312.968,Z 154.498,A -85,B 0,C 180,E1 -15481.287,E2 -15481.287} C_VEL
LIN {X 0,Y 312.688,Z 154.533,A -85,B 0,C 180,E1 -15485.158,E2 -15485.158} C_VEL
LIN {X 0,Y 312.798,Z 154.51,A -85,B 0,C 180,E1 -15487.748,E2 -15487.748} C_VEL
LIN {X 0,Y 312.665,Z 154.532,A -85,B 0,C 180,E1 -15491.672,E2 -15491.672} C_VEL
LIN {X 0,Y 312.67,Z 154.535,A -85,B 0,C 180,E1 -15494.865,E2 -15494.865} C_VEL
LIN {X 0,Y 312.593,Z 154.542,A -85,B 0,C 180,E1 -15499.216,E2 -15499.216} C_VEL
LIN {X 0,Y 312.525,Z 154.543,A -85,B 0,C 180,E1 -15502.779,E2 -15502.779} C_VEL
LIN {X 0,Y 312.532,Z 154.547,A -85,B 0,C 180,E1 -15505.908,E2 -15505.908} C_VEL
LIN {X 0,Y 312.498,Z 154.554,A -85,B 0,C 180,E1 -15509.655,E2 -15509.655} C_VEL
LIN {X 0,Y 312.522,Z 154.55,A -85,B 0,C 180,E1 -15513.689,E2 -15513.689} C_VEL
LIN {X 0,Y 312.516,Z 154.551,A -85,B 0,C 180,E1 -15517.387,E2 -15517.387} C_VEL
LIN {X 0,Y 312.443,Z 154.564,A -85,B 0,C 180,E1 -15520.717,E2 -15520.717} C_VEL
LIN {X 0,Y 312.453,Z 154.568,A -85,B 0,C 180,E1 -15524.21,E2 -15524.21} C_VEL
LIN {X 0,Y 312.486,Z 154.562,A -85,B 0,C 180,E1 -15527.919,E2 -15527.919} C_VEL
LIN {X 0,Y 312.508,Z 154.551,A -85,B 0,C 180,E1 -15531.917,E2 -15531.917} C_VEL
LIN {X 0,Y 312.542,Z 154.754,A -85,B 0,C 180,E1 -15533.784,E2 -15533.784} C_VEL
LIN {X 0,Y 314.981,Z 163.758,A -85,B 0,C 180,E1 -15536.862,E2 -15536.862} C_VEL
LIN {X 0,Y 317.642,Z 175.246,A -85,B 0,C 180,E1 -15540.49,E2 -15540.49} C_VEL
LIN {X 0,Y 318.888,Z 182.236,A -85,B 0,C 180,E1 -15542.505,E2 -15542.505} C_VEL
LIN {X 0,Y 321.186,Z 190.896,A -85,B 0,C 180,E1 -15542.994,E2 -15542.994} C_VEL
LIN {X 0,Y 325.996,Z 215.51,A -85,B 0,C 180,E1 -15544.153,E2 -15544.153} C_VEL
LIN {X 0,Y 327.696,Z 227.543,A -85,B 0,C 180,E1 -15544.637,E2 -15544.637} C_VEL
LIN {X 0,Y 325.895,Z 291.184,A -85,B 0,C 180,E1 -15546.107,E2 -15546.107} C_VEL
LIN {X 0,Y 324.842,Z 305.008,A -85,B 0,C 180,E1 -15546.659,E2 -15546.659} C_VEL
LIN {X 0,Y 323.449,Z 317.46,A -85,B 0,C 180,E1 -15547.398,E2 -15547.398} C_VEL
LIN {X 0,Y 321.797,Z 329.389,A -85,B 0,C 180,E1 -15548.374,E2 -15548.374} C_VEL
LIN {X 0,Y 320.024,Z 340.82,A -85,B 0,C 180,E1 -15549.596,E2 -15549.596} C_VEL
LIN {X 0,Y 318.183,Z 351.16,A -85,B 0,C 180,E1 -15550.986,E2 -15550.986} C_VEL
LIN {X 0,Y 316.331,Z 360.821,A -85,B 0,C 180,E1 -15552.613,E2 -15552.613} C_VEL
LIN {X 0,Y 314.693,Z 369.551,A -85,B 0,C 180,E1 -15554.455,E2 -15554.455} C_VEL
LIN {X 0,Y 313.333,Z 376.883,A -85,B 0,C 180,E1 -15556.378,E2 -15556.378} C_VEL
LIN {X 0,Y 312.131,Z 382.79,A -85,B 0,C 180,E1 -15558.308,E2 -15558.308} C_VEL
LIN {X 0,Y 311.428,Z 387.476,A -85,B 0,C 180,E1 -15560.255,E2 -15560.255} C_VEL
LIN {X 0,Y 310.983,Z 391.074,A -85,B 0,C 180,E1 -15562.207,E2 -15562.207} C_VEL
LIN {X 0,Y 310.728,Z 393.933,A -85,B 0,C 180,E1 -15564.378,E2 -15564.378} C_VEL
LIN {X 0,Y 310.745,Z 395.36,A -85,B 0,C 180,E1 -15566.109,E2 -15566.109} C_VEL
LIN {X 0,Y 310.735,Z 395.991,A -85,B 0,C 180,E1 -15567.407,E2 -15567.407} C_VEL
LIN {X 0,Y 310.775,Z 396.22,A -85,B 0,C 180,E1 -15568.704,E2 -15568.704} C_VEL
LIN {X 0,Y 310.861,Z 396.019,A -85,B 0,C 180,E1 -15570,E2 -15570} C_VEL
LIN {X 0,Y 310.805,Z 395.417,A -85,B 0,C 180,E1 -15571.295,E2 -15571.295} C_VEL
LIN {X 0,Y 310.763,Z 394.42,A -85,B 0,C 180,E1 -15572.592,E2 -15572.592} C_VEL
LIN {X 0,Y 310.785,Z 393.005,A -85,B 0,C 180,E1 -15573.89,E2 -15573.89} C_VEL
LIN {X 0,Y 310.776,Z 390.248,A -85,B 0,C 180,E1 -15575.71,E2 -15575.71} C_VEL
LIN {X 0,Y 310.962,Z 385.974,A -85,B 0,C 180,E1 -15577.793,E2 -15577.793} C_VEL
LIN {X 0,Y 311.388,Z 379.711,A -85,B 0,C 180,E1 -15580.074,E2 -15580.074} C_VEL
LIN {X 0,Y 312.037,Z 372.87,A -85,B 0,C 180,E1 -15582.025,E2 -15582.025} C_VEL
LIN {X 0,Y 312.851,Z 365.892,A -85,B 0,C 180,E1 -15583.643,E2 -15583.643} C_VEL
LIN {X 0,Y 313.795,Z 357.464,A -85,B 0,C 180,E1 -15585.258,E2 -15585.258} C_VEL
LIN {X 0,Y 314.98,Z 347.091,A -85,B 0,C 180,E1 -15586.861,E2 -15586.861} C_VEL
LIN {X 0,Y 316.227,Z 335.355,A -85,B 0,C 180,E1 -15588.295,E2 -15588.295} C_VEL
LIN {X 0,Y 317.463,Z 323.769,A -85,B 0,C 180,E1 -15589.394,E2 -15589.394} C_VEL
LIN {X 0,Y 318.51,Z 311.745,A -85,B 0,C 180,E1 -15590.252,E2 -15590.252} C_VEL
LIN {X 0,Y 319.397,Z 298.777,A -85,B 0,C 180,E1 -15590.908,E2 -15590.908} C_VEL
LIN {X 0,Y 319.866,Z 284.967,A -85,B 0,C 180,E1 -15591.34,E2 -15591.34} C_VEL
LIN {X 0,Y 320.94,Z 224.392,A -85,B 0,C 180,E1 -15592.711,E2 -15592.711} C_VEL
LIN {X 0,Y 315.495,Z 183.275,A -85,B 0,C 180,E1 -15594.049,E2 -15594.049} C_VEL
LIN {X 0,Y 316.411,Z 173.94,A -85,B 0,C 180,E1 -15596.374,E2 -15596.374} C_VEL
LIN {X 0,Y 314.25,Z 162.545,A -85,B 0,C 180,E1 -15599.473,E2 -15599.473} C_VEL
LIN {X 0,Y 312.549,Z 154.553,A -85,B 0,C 180,E1 -15601.75,E2 -15601.75} C_VEL
LIN {X 0,Y 312.537,Z 154.557,A -85,B 0,C 180,E1 -15605.949,E2 -15605.949} C_VEL
LIN {X 0,Y 312.509,Z 154.555,A -85,B 0,C 180,E1 -15609.027,E2 -15609.027} C_VEL
LIN {X 0,Y 312.491,Z 154.558,A -85,B 0,C 180,E1 -15612.431,E2 -15612.431} C_VEL
LIN {X 0,Y 312.459,Z 154.564,A -85,B 0,C 180,E1 -15616.035,E2 -15616.035} C_VEL
LIN {X 0,Y 312.504,Z 154.559,A -85,B 0,C 180,E1 -15619.874,E2 -15619.874} C_VEL
LIN {X 0,Y 312.535,Z 154.553,A -85,B 0,C 180,E1 -15624.05,E2 -15624.05} C_VEL
LIN {X 0,Y 312.504,Z 154.56,A -85,B 0,C 180,E1 -15627.334,E2 -15627.334} C_VEL
LIN {X 0,Y 312.553,Z 154.554,A -85,B 0,C 180,E1 -15631.276,E2 -15631.276} C_VEL
LIN {X 0,Y 312.585,Z 154.546,A -85,B 0,C 180,E1 -15634.711,E2 -15634.711} C_VEL
LIN {X 0,Y 312.564,Z 154.549,A -85,B 0,C 180,E1 -15637.527,E2 -15637.527} C_VEL
LIN {X 0,Y 312.582,Z 154.539,A -85,B 0,C 180,E1 -15641.653,E2 -15641.653} C_VEL
LIN {X 0,Y 312.685,Z 154.531,A -85,B 0,C 180,E1 -15645.686,E2 -15645.686} C_VEL
LIN {X 0,Y 312.685,Z 154.533,A -85,B 0,C 180,E1 -15649.641,E2 -15649.641} C_VEL
LIN {X 0,Y 312.799,Z 154.518,A -85,B 0,C 180,E1 -15652.252,E2 -15652.252} C_VEL
LIN {X 0,Y 312.706,Z 154.533,A -85,B 0,C 180,E1 -15654.842,E2 -15654.842} C_VEL
LIN {X 0,Y 312.988,Z 154.5,A -85,B 0,C 180,E1 -15658.713,E2 -15658.713} C_VEL
LIN {X 0,Y 312.988,Z 154.493,A -85,B 0,C 180,E1 -15661.286,E2 -15661.286} C_VEL
LIN {X 0,Y 312.714,Z 154.529,A -85,B 0,C 180,E1 -15665.157,E2 -15665.157} C_VEL
LIN {X 0,Y 312.852,Z 154.512,A -85,B 0,C 180,E1 -15667.746,E2 -15667.746} C_VEL
LIN {X 0,Y 312.669,Z 154.532,A -85,B 0,C 180,E1 -15671.671,E2 -15671.671} C_VEL
LIN {X 0,Y 312.699,Z 154.532,A -85,B 0,C 180,E1 -15674.887,E2 -15674.887} C_VEL
LIN {X 0,Y 312.608,Z 154.541,A -85,B 0,C 180,E1 -15679.225,E2 -15679.225} C_VEL
LIN {X 0,Y 312.525,Z 154.552,A -85,B 0,C 180,E1 -15682.78,E2 -15682.78} C_VEL
LIN {X 0,Y 312.601,Z 154.547,A -85,B 0,C 180,E1 -15685.935,E2 -15685.935} C_VEL
LIN {X 0,Y 312.537,Z 154.552,A -85,B 0,C 180,E1 -15689.651,E2 -15689.651} C_VEL
LIN {X 0,Y 312.518,Z 154.556,A -85,B 0,C 180,E1 -15693.689,E2 -15693.689} C_VEL
LIN {X 0,Y 312.519,Z 154.554,A -85,B 0,C 180,E1 -15697.386,E2 -15697.386} C_VEL
LIN {X 0,Y 312.489,Z 154.556,A -85,B 0,C 180,E1 -15700.709,E2 -15700.709} C_VEL
LIN {X 0,Y 312.45,Z 154.562,A -85,B 0,C 180,E1 -15704.21,E2 -15704.21} C_VEL
LIN {X 0,Y 312.483,Z 154.56,A -85,B 0,C 180,E1 -15707.919,E2 -15707.919} C_VEL
LIN {X 0,Y 312.504,Z 154.557,A -85,B 0,C 180,E1 -15711.917,E2 -15711.917} C_VEL
LIN {X 0,Y 312.53,Z 154.552,A -85,B 0,C 180,E1 -15714.22,E2 -15714.22} C_VEL
LIN {X 0,Y 312.503,Z 154.558,A -85,B 0,C 180,E1 -15717.334,E2 -15717.334} C_VEL
LIN {X 0,Y 312.551,Z 154.554,A -85,B 0,C 180,E1 -15721.276,E2 -15721.276} C_VEL
LIN {X 0,Y 312.584,Z 154.546,A -85,B 0,C 180,E1 -15724.711,E2 -15724.711} C_VEL
LIN {X 0,Y 312.563,Z 154.55,A -85,B 0,C 180,E1 -15727.527,E2 -15727.527} C_VEL
LIN {X 0,Y 312.581,Z 154.546,A -85,B 0,C 180,E1 -15731.653,E2 -15731.653} C_VEL
LIN {X 0,Y 312.685,Z 154.533,A -85,B 0,C 180,E1 -15735.686,E2 -15735.686} C_VEL
LIN {X 0,Y 312.685,Z 154.534,A -85,B 0,C 180,E1 -15739.642,E2 -15739.642} C_VEL
LIN {X 0,Y 312.799,Z 154.518,A -85,B 0,C 180,E1 -15742.253,E2 -15742.253} C_VEL
LIN {X 0,Y 312.727,Z 154.533,A -85,B 0,C 180,E1 -15745.166,E2 -15745.166} C_VEL
LIN {X 0,Y 313.16,Z 156.92,A -85,B 0,C 180,E1 -15745.898,E2 -15745.898} C_VEL
LIN {X 0,Y 319.165,Z 173.775,A -85,B 0,C 180,E1 -15746.708,E2 -15746.708} C_VEL
LIN {X 0,Y 320.955,Z 180.143,A -85,B 0,C 180,E1 -15746.972,E2 -15746.972} C_VEL
LIN {X 0,Y 321.783,Z 185.585,A -85,B 0,C 180,E1 -15747.152,E2 -15747.152} C_VEL
LIN {X 0,Y 319.988,Z 264.147,A -85,B 0,C 180,E1 -15748.938,E2 -15748.938} C_VEL
LIN {X 0,Y 319.401,Z 277.393,A -85,B 0,C 180,E1 -15749.488,E2 -15749.488} C_VEL
LIN {X 0,Y 318.716,Z 290.61,A -85,B 0,C 180,E1 -15750.316,E2 -15750.316} C_VEL
LIN {X 0,Y 317.825,Z 301.827,A -85,B 0,C 180,E1 -15751.267,E2 -15751.267} C_VEL
LIN {X 0,Y 316.68,Z 313.516,A -85,B 0,C 180,E1 -15752.544,E2 -15752.544} C_VEL
LIN {X 0,Y 315.529,Z 324.037,A -85,B 0,C 180,E1 -15753.992,E2 -15753.992} C_VEL
LIN {X 0,Y 314.498,Z 332.627,A -85,B 0,C 180,E1 -15755.45,E2 -15755.45} C_VEL
LIN {X 0,Y 313.344,Z 341.912,A -85,B 0,C 180,E1 -15757.41,E2 -15757.41} C_VEL
LIN {X 0,Y 312.48,Z 349.375,A -85,B 0,C 180,E1 -15759.385,E2 -15759.385} C_VEL
LIN {X 0,Y 311.898,Z 354.416,A -85,B 0,C 180,E1 -15761.042,E2 -15761.042} C_VEL
LIN {X 0,Y 311.414,Z 359.298,A -85,B 0,C 180,E1 -15763.043,E2 -15763.043} C_VEL
LIN {X 0,Y 311.036,Z 363.029,A -85,B 0,C 180,E1 -15765.061,E2 -15765.061} C_VEL
LIN {X 0,Y 310.75,Z 365.692,A -85,B 0,C 180,E1 -15767.099,E2 -15767.099} C_VEL
LIN {X 0,Y 310.667,Z 366.897,A -85,B 0,C 180,E1 -15768.464,E2 -15768.464} C_VEL
LIN {X 0,Y 310.643,Z 367.645,A -85,B 0,C 180,E1 -15769.838,E2 -15769.838} C_VEL
LIN {X 0,Y 310.765,Z 367.95,A -85,B 0,C 180,E1 -15771.995,E2 -15771.995} C_VEL
LIN {X 0,Y 310.984,Z 367.259,A -85,B 0,C 180,E1 -15774.003,E2 -15774.003} C_VEL
LIN {X 0,Y 311.298,Z 366.197,A -85,B 0,C 180,E1 -15775.438,E2 -15775.438} C_VEL
LIN {X 0,Y 311.862,Z 363.755,A -85,B 0,C 180,E1 -15777.515,E2 -15777.515} C_VEL
LIN {X 0,Y 312.698,Z 360.113,A -85,B 0,C 180,E1 -15779.634,E2 -15779.634} C_VEL
LIN {X 0,Y 313.891,Z 354.497,A -85,B 0,C 180,E1 -15781.99,E2 -15781.99} C_VEL
LIN {X 0,Y 315.404,Z 347.52,A -85,B 0,C 180,E1 -15784.209,E2 -15784.209} C_VEL
LIN {X 0,Y 316.9,Z 340.376,A -85,B 0,C 180,E1 -15785.994,E2 -15785.994} C_VEL
LIN {X 0,Y 318.682,Z 330.988,A -85,B 0,C 180,E1 -15787.87,E2 -15787.87} C_VEL
LIN {X 0,Y 320.56,Z 320.847,A -85,B 0,C 180,E1 -15789.48,E2 -15789.48} C_VEL
LIN {X 0,Y 322.326,Z 309.851,A -85,B 0,C 180,E1 -15790.853,E2 -15790.853} C_VEL
LIN {X 0,Y 323.963,Z 297.587,A -85,B 0,C 180,E1 -15792.052,E2 -15792.052} C_VEL
LIN {X 0,Y 325.193,Z 285.16,A -85,B 0,C 180,E1 -15792.969,E2 -15792.969} C_VEL
LIN {X 0,Y 326.173,Z 272.15,A -85,B 0,C 180,E1 -15793.641,E2 -15793.641} C_VEL
LIN {X 0,Y 326.738,Z 259.645,A -85,B 0,C 180,E1 -15794.052,E2 -15794.052} C_VEL
LIN {X 0,Y 328.342,Z 204.966,A -85,B 0,C 180,E1 -15795.288,E2 -15795.288} C_VEL
LIN {X 0,Y 328.025,Z 201.131,A -85,B 0,C 180,E1 -15795.42,E2 -15795.42} C_VEL
LIN {X 0,Y 326.38,Z 195.728,A -85,B 0,C 180,E1 -15795.731,E2 -15795.731} C_VEL
LIN {X 0,Y 323.864,Z 190.79,A -85,B 0,C 180,E1 -15796.129,E2 -15796.129} C_VEL
LIN {X 0,Y 316.128,Z 177.812,A -85,B 0,C 180,E1 -15797.343,E2 -15797.343} C_VEL
LIN {X 0,Y 309.409,Z 164.747,A -85,B 0,C 180,E1 -15798.514,E2 -15798.514} C_VEL
LIN {X 0,Y 306.264,Z 158.743,A -85,B 0,C 180,E1 -15799.093,E2 -15799.093} C_VEL
LIN {X 0,Y 305.418,Z 155.435,A -85,B 0,C 180,E1 -15800.423,E2 -15800.423} C_VEL
LIN {X 0,Y 305.461,Z 155.423,A -85,B 0,C 180,E1 -15803.637,E2 -15803.637} C_VEL
LIN {X 0,Y 305.465,Z 155.434,A -85,B 0,C 180,E1 -15806.483,E2 -15806.483} C_VEL
LIN {X 0,Y 305.418,Z 155.445,A -85,B 0,C 180,E1 -15809.586,E2 -15809.586} C_VEL
LIN {X 0,Y 305.441,Z 155.442,A -85,B 0,C 180,E1 -15812.601,E2 -15812.601} C_VEL
LIN {X 0,Y 305.44,Z 155.44,A -85,B 0,C 180,E1 -15815.533,E2 -15815.533} C_VEL
LIN {X 0,Y 305.474,Z 155.435,A -85,B 0,C 180,E1 -15819.812,E2 -15819.812} C_VEL
LIN {X 0,Y 305.493,Z 155.428,A -85,B 0,C 180,E1 -15823.975,E2 -15823.975} C_VEL
LIN {X 0,Y 305.555,Z 155.425,A -85,B 0,C 180,E1 -15826.703,E2 -15826.703} C_VEL
LIN {X 0,Y 305.755,Z 155.397,A -85,B 0,C 180,E1 -15831.261,E2 -15831.261} C_VEL
LIN {X 0,Y 305.786,Z 155.383,A -85,B 0,C 180,E1 -15833.401,E2 -15833.401} C_VEL
LIN {X 0,Y 305.935,Z 155.365,A -85,B 0,C 180,E1 -15838.684,E2 -15838.684} C_VEL
LIN {X 0,Y 305.936,Z 155.374,A -85,B 0,C 180,E1 -15841.317,E2 -15841.317} C_VEL
LIN {X 0,Y 305.787,Z 155.39,A -85,B 0,C 180,E1 -15846.599,E2 -15846.599} C_VEL
LIN {X 0,Y 305.696,Z 155.4,A -85,B 0,C 180,E1 -15849.261,E2 -15849.261} C_VEL
LIN {X 0,Y 305.588,Z 155.408,A -85,B 0,C 180,E1 -15853.296,E2 -15853.296} C_VEL
LIN {X 0,Y 305.553,Z 155.421,A -85,B 0,C 180,E1 -15856.023,E2 -15856.023} C_VEL
LIN {X 0,Y 305.549,Z 155.422,A -85,B 0,C 180,E1 -15859.429,E2 -15859.429} C_VEL
LIN {X 0,Y 305.488,Z 155.422,A -85,B 0,C 180,E1 -15863.039,E2 -15863.039} C_VEL
LIN {X 0,Y 305.472,Z 155.424,A -85,B 0,C 180,E1 -15866.197,E2 -15866.197} C_VEL
LIN {X 0,Y 305.451,Z 155.436,A -85,B 0,C 180,E1 -15869.034,E2 -15869.034} C_VEL
LIN {X 0,Y 305.439,Z 155.437,A -85,B 0,C 180,E1 -15871.953,E2 -15871.953} C_VEL
LIN {X 0,Y 305.464,Z 155.433,A -85,B 0,C 180,E1 -15875.113,E2 -15875.113} C_VEL
LIN {X 0,Y 305.435,Z 155.438,A -85,B 0,C 180,E1 -15878.525,E2 -15878.525} C_VEL
LIN {X 0,Y 305.438,Z 155.439,A -85,B 0,C 180,E1 -15882.582,E2 -15882.582} C_VEL
LIN {X 0,Y 305.428,Z 155.442,A -85,B 0,C 180,E1 -15886.345,E2 -15886.345} C_VEL
LIN {X 0,Y 305.46,Z 155.436,A -85,B 0,C 180,E1 -15889.892,E2 -15889.892} C_VEL
LIN {X 0,Y 305.505,Z 155.449,A -85,B 0,C 180,E1 -15892.955,E2 -15892.955} C_VEL
LIN {X 0,Y 307.845,Z 164.264,A -85,B 0,C 180,E1 -15896.07,E2 -15896.07} C_VEL
LIN {X 0,Y 310.459,Z 175.271,A -85,B 0,C 180,E1 -15899.697,E2 -15899.697} C_VEL
LIN {X 0,Y 311.803,Z 181.858,A -85,B 0,C 180,E1 -15901.669,E2 -15901.669} C_VEL
LIN {X 0,Y 314.247,Z 188.478,A -85,B 0,C 180,E1 -15902.14,E2 -15902.14} C_VEL
